LIN {X 0,Y 388.743,Z 625.918,A -85,B 0,C 180,E1 -11613.109,E2 -11613.109} C_VEL
LIN {X 0,Y 388.739,Z 624.507,A -85,B 0,C 180,E1 -11614.147,E2 -11614.147} C_VEL
LIN {X 0,Y 388.741,Z 621.416,A -85,B 0,C 180,E1 -11615.775,E2 -11615.775} C_VEL
LIN {X 0,Y 388.932,Z 617.582,A -85,B 0,C 180,E1 -11617.267,E2 -11617.267} C_VEL
LIN {X 0,Y 389.218,Z 612.461,A -85,B 0,C 180,E1 -11618.829,E2 -11618.829} C_VEL
LIN {X 0,Y 389.638,Z 606.07,A -85,B 0,C 180,E1 -11620.392,E2 -11620.392} C_VEL
LIN {X 0,Y 390.339,Z 598.224,A -85,B 0,C 180,E1 -11621.95,E2 -11621.95} C_VEL
LIN {X 0,Y 391.121,Z 588.53,A -85,B 0,C 180,E1 -11623.509,E2 -11623.509} C_VEL
LIN {X 0,Y 392.289,Z 577.655,A -85,B 0,C 180,E1 -11624.924,E2 -11624.924} C_VEL
LIN {X 0,Y 393.398,Z 566.699,A -85,B 0,C 180,E1 -11626.076,E2 -11626.076} C_VEL
LIN {X 0,Y 394.452,Z 554.774,A -85,B 0,C 180,E1 -11627.097,E2 -11627.097} C_VEL
LIN {X 0,Y 393.842,Z 541.578,A -85,B 0,C 180,E1 -11628.085,E2 -11628.085} C_VEL
LIN {X 0,Y 392.175,Z 529.359,A -85,B 0,C 180,E1 -11628.886,E2 -11628.886} C_VEL
LIN {X 0,Y 389.451,Z 517.138,A -85,B 0,C 180,E1 -11629.64,E2 -11629.64} C_VEL
LIN {X 0,Y 389.818,Z 510.265,A -85,B 0,C 180,E1 -11632.714,E2 -11632.714} C_VEL
LIN {X 0,Y 390.359,Z 503.675,A -85,B 0,C 180,E1 -11635.816,E2 -11635.816} C_VEL
LIN {X 0,Y 391.097,Z 496.234,A -85,B 0,C 180,E1 -11639.615,E2 -11639.615} C_VEL
LIN {X 0,Y 391.871,Z 491.031,A -85,B 0,C 180,E1 -11642.55,E2 -11642.55} C_VEL
LIN {X 0,Y 392.449,Z 487.212,A -85,B 0,C 180,E1 -11644.964,E2 -11644.964} C_VEL
LIN {X 0,Y 392.679,Z 485.233,A -85,B 0,C 180,E1 -11646.352,E2 -11646.352} C_VEL
LIN {X 0,Y 392.542,Z 482.258,A -85,B 0,C 180,E1 -11648.802,E2 -11648.802} C_VEL
LIN {X 0,Y 392.126,Z 479.631,A -85,B 0,C 180,E1 -11651.54,E2 -11651.54} C_VEL
LIN {X 0,Y 391.771,Z 477.585,A -85,B 0,C 180,E1 -11654.397,E2 -11654.397} C_VEL
LIN {X 0,Y 391.509,Z 476.207,A -85,B 0,C 180,E1 -11657.391,E2 -11657.391} C_VEL
LIN {X 0,Y 391.301,Z 475.518,A -85,B 0,C 180,E1 -11660.562,E2 -11660.562} C_VEL
LIN {X 0,Y 391.175,Z 475.523,A -85,B 0,C 180,E1 -11663.638,E2 -11663.638} C_VEL
LIN {X 0,Y 390.977,Z 475.957,A -85,B 0,C 180,E1 -11666.135,E2 -11666.135} C_VEL
LIN {X 0,Y 390.563,Z 477.165,A -85,B 0,C 180,E1 -11669.745,E2 -11669.745} C_VEL
LIN {X 0,Y 390.158,Z 478.822,A -85,B 0,C 180,E1 -11673.235,E2 -11673.235} C_VEL
LIN {X 0,Y 389.91,Z 480.896,A -85,B 0,C 180,E1 -11676.819,E2 -11676.819} C_VEL
LIN {X 0,Y 389.699,Z 483.382,A -85,B 0,C 180,E1 -11680.549,E2 -11680.549} C_VEL
LIN {X 0,Y 394.387,Z 496.846,A -85,B 0,C 180,E1 -11681.609,E2 -11681.609} C_VEL
LIN {X 0,Y 396.401,Z 504.348,A -85,B 0,C 180,E1 -11682.226,E2 -11682.226} C_VEL
LIN {X 0,Y 396.513,Z 507.54,A -85,B 0,C 180,E1 -11682.463,E2 -11682.463} C_VEL
LIN {X 0,Y 395.554,Z 519.166,A -85,B 0,C 180,E1 -11683.352,E2 -11683.352} C_VEL
LIN {X 0,Y 394.437,Z 530.942,A -85,B 0,C 180,E1 -11684.498,E2 -11684.498} C_VEL
LIN {X 0,Y 393.337,Z 541.589,A -85,B 0,C 180,E1 -11685.778,E2 -11685.778} C_VEL
LIN {X 0,Y 392.489,Z 548.688,A -85,B 0,C 180,E1 -11686.803,E2 -11686.803} C_VEL
LIN {X 0,Y 391.496,Z 557.528,A -85,B 0,C 180,E1 -11688.349,E2 -11688.349} C_VEL
LIN {X 0,Y 390.789,Z 564.646,A -85,B 0,C 180,E1 -11689.901,E2 -11689.901} C_VEL
LIN {X 0,Y 390.054,Z 571.233,A -85,B 0,C 180,E1 -11691.712,E2 -11691.712} C_VEL
LIN {X 0,Y 389.636,Z 575.213,A -85,B 0,C 180,E1 -11693.115,E2 -11693.115} C_VEL
LIN {X 0,Y 389.321,Z 578.854,A -85,B 0,C 180,E1 -11694.822,E2 -11694.822} C_VEL
LIN {X 0,Y 389.232,Z 580.45,A -85,B 0,C 180,E1 -11695.858,E2 -11695.858} C_VEL
LIN {X 0,Y 389.059,Z 581.651,A -85,B 0,C 180,E1 -11696.894,E2 -11696.894} C_VEL
LIN {X 0,Y 388.959,Z 582.45,A -85,B 0,C 180,E1 -11697.929,E2 -11697.929} C_VEL
LIN {X 0,Y 388.866,Z 582.808,A -85,B 0,C 180,E1 -11698.965,E2 -11698.965} C_VEL
LIN {X 0,Y 388.812,Z 582.757,A -85,B 0,C 180,E1 -11700,E2 -11700} C_VEL
LIN {X 0,Y 388.817,Z 582.311,A -85,B 0,C 180,E1 -11701.036,E2 -11701.036} C_VEL
LIN {X 0,Y 388.9,Z 581.459,A -85,B 0,C 180,E1 -11702.072,E2 -11702.072} C_VEL
LIN {X 0,Y 388.979,Z 580.155,A -85,B 0,C 180,E1 -11703.107,E2 -11703.107} C_VEL
LIN {X 0,Y 388.992,Z 577.422,A -85,B 0,C 180,E1 -11704.664,E2 -11704.664} C_VEL
LIN {X 0,Y 389.28,Z 572.842,A -85,B 0,C 180,E1 -11706.498,E2 -11706.498} C_VEL
LIN {X 0,Y 389.595,Z 566.823,A -85,B 0,C 180,E1 -11708.298,E2 -11708.298} C_VEL
LIN {X 0,Y 390.104,Z 560.131,A -85,B 0,C 180,E1 -11709.855,E2 -11709.855} C_VEL
LIN {X 0,Y 390.663,Z 551.845,A -85,B 0,C 180,E1 -11711.414,E2 -11711.414} C_VEL
LIN {X 0,Y 391.294,Z 543.426,A -85,B 0,C 180,E1 -11712.711,E2 -11712.711} C_VEL
LIN {X 0,Y 392.117,Z 533.146,A -85,B 0,C 180,E1 -11714.003,E2 -11714.003} C_VEL
LIN {X 0,Y 392.805,Z 521.468,A -85,B 0,C 180,E1 -11715.191,E2 -11715.191} C_VEL
LIN {X 0,Y 393.462,Z 510.623,A -85,B 0,C 180,E1 -11716.073,E2 -11716.073} C_VEL
LIN {X 0,Y 393.827,Z 501.011,A -85,B 0,C 180,E1 -11716.706,E2 -11716.706} C_VEL
LIN {X 0,Y 391.065,Z 488.304,A -85,B 0,C 180,E1 -11717.466,E2 -11717.466} C_VEL
LIN {X 0,Y 388.963,Z 478.596,A -85,B 0,C 180,E1 -11717.923,E2 -11717.923} C_VEL
LIN {X 0,Y 389.004,Z 475.238,A -85,B 0,C 180,E1 -11721.182,E2 -11721.182} C_VEL
LIN {X 0,Y 389.069,Z 471.846,A -85,B 0,C 180,E1 -11724.549,E2 -11724.549} C_VEL
LIN {X 0,Y 389.216,Z 468.447,A -85,B 0,C 180,E1 -11728.001,E2 -11728.001} C_VEL
LIN {X 0,Y 389.39,Z 467.987,A -85,B 0,C 180,E1 -11729.963,E2 -11729.963} C_VEL
LIN {X 0,Y 389.666,Z 467.948,A -85,B 0,C 180,E1 -11732.758,E2 -11732.758} C_VEL
LIN {X 0,Y 389.974,Z 467.908,A -85,B 0,C 180,E1 -11735.808,E2 -11735.808} C_VEL
LIN {X 0,Y 390.07,Z 467.894,A -85,B 0,C 180,E1 -11739.218,E2 -11739.218} C_VEL
LIN {X 0,Y 390.049,Z 467.9,A -85,B 0,C 180,E1 -11742.375,E2 -11742.375} C_VEL
LIN {X 0,Y 390.05,Z 467.897,A -85,B 0,C 180,E1 -11745.355,E2 -11745.355} C_VEL
LIN {X 0,Y 390.036,Z 467.902,A -85,B 0,C 180,E1 -11748.187,E2 -11748.187} C_VEL
LIN {X 0,Y 390.097,Z 467.891,A -85,B 0,C 180,E1 -11750.908,E2 -11750.908} C_VEL
LIN {X 0,Y 390.089,Z 467.892,A -85,B 0,C 180,E1 -11754.793,E2 -11754.793} C_VEL
LIN {X 0,Y 390.036,Z 467.902,A -85,B 0,C 180,E1 -11757.875,E2 -11757.875} C_VEL
LIN {X 0,Y 390.063,Z 467.896,A -85,B 0,C 180,E1 -11760.891,E2 -11760.891} C_VEL
LIN {X 0,Y 390.124,Z 467.893,A -85,B 0,C 180,E1 -11764.257,E2 -11764.257} C_VEL
LIN {X 0,Y 390.045,Z 467.9,A -85,B 0,C 180,E1 -11767.766,E2 -11767.766} C_VEL
LIN {X 0,Y 390.11,Z 467.89,A -85,B 0,C 180,E1 -11771.078,E2 -11771.078} C_VEL
LIN {X 0,Y 390.144,Z 467.889,A -85,B 0,C 180,E1 -11774.323,E2 -11774.323} C_VEL
LIN {X 0,Y 390.176,Z 467.882,A -85,B 0,C 180,E1 -11777.517,E2 -11777.517} C_VEL
LIN {X 0,Y 390.32,Z 467.866,A -85,B 0,C 180,E1 -11781.718,E2 -11781.718} C_VEL
LIN {X 0,Y 390.335,Z 467.865,A -85,B 0,C 180,E1 -11783.798,E2 -11783.798} C_VEL
LIN {X 0,Y 390.423,Z 467.853,A -85,B 0,C 180,E1 -11787.937,E2 -11787.937} C_VEL
LIN {X 0,Y 390.554,Z 467.838,A -85,B 0,C 180,E1 -11790,E2 -11790} C_VEL
LIN {X 0,Y 390.315,Z 467.863,A -85,B 0,C 180,E1 -11793.097,E2 -11793.097} C_VEL
LIN {X 0,Y 390.304,Z 467.868,A -85,B 0,C 180,E1 -11796.202,E2 -11796.202} C_VEL
LIN {X 0,Y 390.198,Z 467.88,A -85,B 0,C 180,E1 -11799.329,E2 -11799.329} C_VEL
LIN {X 0,Y 390.176,Z 467.882,A -85,B 0,C 180,E1 -11802.483,E2 -11802.483} C_VEL
LIN {X 0,Y 390.145,Z 467.888,A -85,B 0,C 180,E1 -11805.677,E2 -11805.677} C_VEL
LIN {X 0,Y 390.111,Z 467.89,A -85,B 0,C 180,E1 -11808.922,E2 -11808.922} C_VEL
LIN {X 0,Y 390.041,Z 467.9,A -85,B 0,C 180,E1 -11812.32,E2 -11812.32} C_VEL
LIN {X 0,Y 390.123,Z 467.891,A -85,B 0,C 180,E1 -11815.743,E2 -11815.743} C_VEL
LIN {X 0,Y 390.115,Z 467.887,A -85,B 0,C 180,E1 -11816.807,E2 -11816.807} C_VEL
LIN {X 0,Y 389.411,Z 467.98,A -85,B 0,C 180,E1 -11817.668,E2 -11817.668} C_VEL
LIN {X 0,Y 386.517,Z 468.337,A -85,B 0,C 180,E1 -11819.069,E2 -11819.069} C_VEL
LIN {X 0,Y 384.091,Z 468.642,A -85,B 0,C 180,E1 -11820.2,E2 -11820.2} C_VEL
LIN {X 0,Y 383.057,Z 468.768,A -85,B 0,C 180,E1 -11821.076,E2 -11821.076} C_VEL
LIN {X 0,Y 382.977,Z 468.777,A -85,B 0,C 180,E1 -11821.372,E2 -11821.372} C_VEL
LIN {X 0,Y 383.023,Z 468.772,A -85,B 0,C 180,E1 -11824.668,E2 -11824.668} C_VEL
LIN {X 0,Y 383.006,Z 468.778,A -85,B 0,C 180,E1 -11827.904,E2 -11827.904} C_VEL
LIN {X 0,Y 382.989,Z 468.778,A -85,B 0,C 180,E1 -11831.347,E2 -11831.347} C_VEL
LIN {X 0,Y 383.001,Z 468.777,A -85,B 0,C 180,E1 -11834.303,E2 -11834.303} C_VEL
LIN {X 0,Y 383.014,Z 468.775,A -85,B 0,C 180,E1 -11837.24,E2 -11837.24} C_VEL
LIN {X 0,Y 383.018,Z 468.772,A -85,B 0,C 180,E1 -11840.413,E2 -11840.413} C_VEL
LIN {X 0,Y 382.973,Z 468.78,A -85,B 0,C 180,E1 -11844.038,E2 -11844.038} C_VEL
LIN {X 0,Y 382.774,Z 468.804,A -85,B 0,C 180,E1 -11846.576,E2 -11846.576} C_VEL
LIN {X 0,Y 382.417,Z 468.852,A -85,B 0,C 180,E1 -11849.742,E2 -11849.742} C_VEL
LIN {X 0,Y 382.061,Z 468.898,A -85,B 0,C 180,E1 -11852.621,E2 -11852.621} C_VEL
LIN {X 0,Y 381.965,Z 469.45,A -85,B 0,C 180,E1 -11853.794,E2 -11853.794} C_VEL
LIN {X 0,Y 381.906,Z 473.282,A -85,B 0,C 180,E1 -11857.266,E2 -11857.266} C_VEL
LIN {X 0,Y 381.87,Z 477.054,A -85,B 0,C 180,E1 -11860.653,E2 -11860.653} C_VEL
LIN {X 0,Y 381.871,Z 478.605,A -85,B 0,C 180,E1 -11861.963,E2 -11861.963} C_VEL
LIN {X 0,Y 384.636,Z 491.634,A -85,B 0,C 180,E1 -11862.594,E2 -11862.594} C_VEL
LIN {X 0,Y 386.939,Z 502.891,A -85,B 0,C 180,E1 -11863.309,E2 -11863.309} C_VEL
LIN {X 0,Y 386.237,Z 514.849,A -85,B 0,C 180,E1 -11864.16,E2 -11864.16} C_VEL
LIN {X 0,Y 385.572,Z 526.535,A -85,B 0,C 180,E1 -11865.215,E2 -11865.215} C_VEL
LIN {X 0,Y 384.771,Z 537.046,A -85,B 0,C 180,E1 -11866.398,E2 -11866.398} C_VEL
LIN {X 0,Y 383.944,Z 547.495,A -85,B 0,C 180,E1 -11867.848,E2 -11867.848} C_VEL
LIN {X 0,Y 383.25,Z 556.654,A -85,B 0,C 180,E1 -11869.433,E2 -11869.433} C_VEL
LIN {X 0,Y 382.693,Z 564.046,A -85,B 0,C 180,E1 -11871.019,E2 -11871.019} C_VEL
LIN {X 0,Y 382.348,Z 570,A -85,B 0,C 180,E1 -11872.607,E2 -11872.607} C_VEL
LIN {X 0,Y 382.089,Z 574.685,A -85,B 0,C 180,E1 -11874.193,E2 -11874.193} C_VEL
LIN {X 0,Y 381.872,Z 578.249,A -85,B 0,C 180,E1 -11875.778,E2 -11875.778} C_VEL
LIN {X 0,Y 381.88,Z 580.026,A -85,B 0,C 180,E1 -11876.835,E2 -11876.835} C_VEL
LIN {X 0,Y 381.827,Z 581.4,A -85,B 0,C 180,E1 -11877.89,E2 -11877.89} C_VEL
LIN {X 0,Y 381.737,Z 582.371,A -85,B 0,C 180,E1 -11878.945,E2 -11878.945} C_VEL
LIN {X 0,Y 381.727,Z 582.881,A -85,B 0,C 180,E1 -11880,E2 -11880} C_VEL
LIN {X 0,Y 381.771,Z 582.992,A -85,B 0,C 180,E1 -11881.055,E2 -11881.055} C_VEL
LIN {X 0,Y 381.875,Z 582.707,A -85,B 0,C 180,E1 -11882.109,E2 -11882.109} C_VEL
LIN {X 0,Y 382.006,Z 581.987,A -85,B 0,C 180,E1 -11883.164,E2 -11883.164} C_VEL
LIN {X 0,Y 382.177,Z 580.837,A -85,B 0,C 180,E1 -11884.218,E2 -11884.218} C_VEL
LIN {X 0,Y 382.189,Z 579.305,A -85,B 0,C 180,E1 -11885.275,E2 -11885.275} C_VEL
LIN {X 0,Y 382.572,Z 576.053,A -85,B 0,C 180,E1 -11886.903,E2 -11886.903} C_VEL
LIN {X 0,Y 382.999,Z 571.944,A -85,B 0,C 180,E1 -11888.441,E2 -11888.441} C_VEL
LIN {X 0,Y 383.807,Z 565.49,A -85,B 0,C 180,E1 -11890.284,E2 -11890.284} C_VEL
LIN {X 0,Y 384.51,Z 558.499,A -85,B 0,C 180,E1 -11891.866,E2 -11891.866} C_VEL
LIN {X 0,Y 385.567,Z 549.85,A -85,B 0,C 180,E1 -11893.438,E2 -11893.438} C_VEL
LIN {X 0,Y 386.583,Z 541.045,A -85,B 0,C 180,E1 -11894.745,E2 -11894.745} C_VEL
LIN {X 0,Y 387.837,Z 530.124,A -85,B 0,C 180,E1 -11896.065,E2 -11896.065} C_VEL
LIN {X 0,Y 389.023,Z 518.194,A -85,B 0,C 180,E1 -11897.207,E2 -11897.207} C_VEL
LIN {X 0,Y 389.929,Z 506.361,A -85,B 0,C 180,E1 -11898.116,E2 -11898.116} C_VEL
LIN {X 0,Y 387.401,Z 496.099,A -85,B 0,C 180,E1 -11898.999,E2 -11898.999} C_VEL
LIN {X 0,Y 383.296,Z 484.971,A -85,B 0,C 180,E1 -11899.92,E2 -11899.92} C_VEL
LIN {X 0,Y 382.567,Z 482.635,A -85,B 0,C 180,E1 -11900.107,E2 -11900.107} C_VEL
LIN {X 0,Y 382.645,Z 478.78,A -85,B 0,C 180,E1 -11903.833,E2 -11903.833} C_VEL
LIN {X 0,Y 382.729,Z 476.402,A -85,B 0,C 180,E1 -11906.149,E2 -11906.149} C_VEL
LIN {X 0,Y 382.822,Z 472.719,A -85,B 0,C 180,E1 -11909.714,E2 -11909.714} C_VEL
LIN {X 0,Y 382.879,Z 470.008,A -85,B 0,C 180,E1 -11912.396,E2 -11912.396} C_VEL
LIN {X 0,Y 382.808,Z 469.012,A -85,B 0,C 180,E1 -11913.42,E2 -11913.42} C_VEL
LIN {X 0,Y 382.987,Z 468.78,A -85,B 0,C 180,E1 -11916.155,E2 -11916.155} C_VEL
LIN {X 0,Y 383.017,Z 468.778,A -85,B 0,C 180,E1 -11919.587,E2 -11919.587} C_VEL
LIN {X 0,Y 383.006,Z 468.777,A -85,B 0,C 180,E1 -11922.778,E2 -11922.778} C_VEL
LIN {X 0,Y 383.057,Z 468.821,A -85,B 0,C 180,E1 -11926.355,E2 -11926.355} C_VEL
LIN {X 0,Y 384.052,Z 474.383,A -85,B 0,C 180,E1 -11929.486,E2 -11929.486} C_VEL
LIN {X 0,Y 385.125,Z 480.888,A -85,B 0,C 180,E1 -11932.972,E2 -11932.972} C_VEL
LIN {X 0,Y 385.096,Z 485.339,A -85,B 0,C 180,E1 -11935.21,E2 -11935.21} C_VEL
LIN {X 0,Y 384.35,Z 492.339,A -85,B 0,C 180,E1 -11938.591,E2 -11938.591} C_VEL
LIN {X 0,Y 383.676,Z 499.918,A -85,B 0,C 180,E1 -11942.154,E2 -11942.154} C_VEL
LIN {X 0,Y 383.037,Z 507.462,A -85,B 0,C 180,E1 -11945.617,E2 -11945.617} C_VEL
LIN {X 0,Y 382.543,Z 514.974,A -85,B 0,C 180,E1 -11949.007,E2 -11949.007} C_VEL
LIN {X 0,Y 382.39,Z 517.633,A -85,B 0,C 180,E1 -11950.192,E2 -11950.192} C_VEL
LIN {X 0,Y 385.614,Z 533.963,A -85,B 0,C 180,E1 -11951.245,E2 -11951.245} C_VEL
LIN {X 0,Y 386.776,Z 546.578,A -85,B 0,C 180,E1 -11952.144,E2 -11952.144} C_VEL
LIN {X 0,Y 387.184,Z 556.631,A -85,B 0,C 180,E1 -11952.981,E2 -11952.981} C_VEL
LIN {X 0,Y 386.052,Z 567.959,A -85,B 0,C 180,E1 -11954.017,E2 -11954.017} C_VEL
LIN {X 0,Y 384.872,Z 579.687,A -85,B 0,C 180,E1 -11955.356,E2 -11955.356} C_VEL
LIN {X 0,Y 383.891,Z 589.69,A -85,B 0,C 180,E1 -11956.771,E2 -11956.771} C_VEL
LIN {X 0,Y 383.004,Z 598.767,A -85,B 0,C 180,E1 -11958.355,E2 -11958.355} C_VEL
LIN {X 0,Y 382.388,Z 606.219,A -85,B 0,C 180,E1 -11959.944,E2 -11959.944} C_VEL
LIN {X 0,Y 382.02,Z 612.209,A -85,B 0,C 180,E1 -11961.537,E2 -11961.537} C_VEL
LIN {X 0,Y 381.745,Z 618.814,A -85,B 0,C 180,E1 -11963.801,E2 -11963.801} C_VEL
LIN {X 0,Y 381.747,Z 622.148,A -85,B 0,C 180,E1 -11965.248,E2 -11965.248} C_VEL
LIN {X 0,Y 381.688,Z 624.791,A -85,B 0,C 180,E1 -11966.833,E2 -11966.833} C_VEL
LIN {X 0,Y 381.779,Z 626.012,A -85,B 0,C 180,E1 -11967.89,E2 -11967.89} C_VEL
LIN {X 0,Y 381.739,Z 626.785,A -85,B 0,C 180,E1 -11968.945,E2 -11968.945} C_VEL
LIN {X 0,Y 381.736,Z 627.103,A -85,B 0,C 180,E1 -11970,E2 -11970} C_VEL
LIN {X 0,Y 381.731,Z 627.012,A -85,B 0,C 180,E1 -11971.055,E2 -11971.055} C_VEL
LIN {X 0,Y 381.756,Z 626.514,A -85,B 0,C 180,E1 -11972.11,E2 -11972.11} C_VEL
LIN {X 0,Y 381.646,Z 625.564,A -85,B 0,C 180,E1 -11973.167,E2 -11973.167} C_VEL
LIN {X 0,Y 381.662,Z 624.175,A -85,B 0,C 180,E1 -11974.224,E2 -11974.224} C_VEL
LIN {X 0,Y 381.693,Z 620.602,A -85,B 0,C 180,E1 -11976.127,E2 -11976.127} C_VEL
LIN {X 0,Y 381.937,Z 615.822,A -85,B 0,C 180,E1 -11977.933,E2 -11977.933} C_VEL
LIN {X 0,Y 382.36,Z 609.307,A -85,B 0,C 180,E1 -11979.789,E2 -11979.789} C_VEL
LIN {X 0,Y 382.939,Z 602.299,A -85,B 0,C 180,E1 -11981.379,E2 -11981.379} C_VEL
LIN {X 0,Y 383.775,Z 593.737,A -85,B 0,C 180,E1 -11982.964,E2 -11982.964} C_VEL
LIN {X 0,Y 384.666,Z 584.669,A -85,B 0,C 180,E1 -11984.336,E2 -11984.336} C_VEL
LIN {X 0,Y 385.946,Z 573.519,A -85,B 0,C 180,E1 -11985.716,E2 -11985.716} C_VEL
LIN {X 0,Y 387.25,Z 561.84,A -85,B 0,C 180,E1 -11986.881,E2 -11986.881} C_VEL
LIN {X 0,Y 387.697,Z 554.173,A -85,B 0,C 180,E1 -11987.54,E2 -11987.54} C_VEL
LIN {X 0,Y 387.066,Z 540.9,A -85,B 0,C 180,E1 -11988.569,E2 -11988.569} C_VEL
LIN {X 0,Y 385.33,Z 529.072,A -85,B 0,C 180,E1 -11989.391,E2 -11989.391} C_VEL
LIN {X 0,Y 382.474,Z 516.569,A -85,B 0,C 180,E1 -11990.191,E2 -11990.191} C_VEL
LIN {X 0,Y 382.931,Z 508.781,A -85,B 0,C 180,E1 -11993.814,E2 -11993.814} C_VEL
LIN {X 0,Y 383.556,Z 501.826,A -85,B 0,C 180,E1 -11997.264,E2 -11997.264} C_VEL
LIN {X 0,Y 384.247,Z 496.405,A -85,B 0,C 180,E1 -12000.178,E2 -12000.178} C_VEL
LIN {X 0,Y 385.024,Z 491.301,A -85,B 0,C 180,E1 -12003.203,E2 -12003.203} C_VEL
LIN {X 0,Y 385.577,Z 487.602,A -85,B 0,C 180,E1 -12005.681,E2 -12005.681} C_VEL
LIN {X 0,Y 385.743,Z 485.902,A -85,B 0,C 180,E1 -12006.959,E2 -12006.959} C_VEL
LIN {X 0,Y 385.677,Z 484.182,A -85,B 0,C 180,E1 -12008.412,E2 -12008.412} C_VEL
LIN {X 0,Y 385.195,Z 481.144,A -85,B 0,C 180,E1 -12011.578,E2 -12011.578} C_VEL
LIN {X 0,Y 384.824,Z 479.04,A -85,B 0,C 180,E1 -12014.581,E2 -12014.581} C_VEL
LIN {X 0,Y 384.587,Z 477.73,A -85,B 0,C 180,E1 -12017.457,E2 -12017.457} C_VEL
LIN {X 0,Y 384.373,Z 477.075,A -85,B 0,C 180,E1 -12020.212,E2 -12020.212} C_VEL
LIN {X 0,Y 384.25,Z 476.956,A -85,B 0,C 180,E1 -12023.588,E2 -12023.588} C_VEL
LIN {X 0,Y 383.928,Z 477.492,A -85,B 0,C 180,E1 -12026.69,E2 -12026.69} C_VEL
LIN {X 0,Y 383.631,Z 478.356,A -85,B 0,C 180,E1 -12029.432,E2 -12029.432} C_VEL
LIN {X 0,Y 383.22,Z 479.79,A -85,B 0,C 180,E1 -12032.711,E2 -12032.711} C_VEL
LIN {X 0,Y 382.928,Z 481.668,A -85,B 0,C 180,E1 -12036.186,E2 -12036.186} C_VEL
LIN {X 0,Y 382.708,Z 484.076,A -85,B 0,C 180,E1 -12039.983,E2 -12039.983} C_VEL
LIN {X 0,Y 383.889,Z 487.251,A -85,B 0,C 180,E1 -12040.241,E2 -12040.241} C_VEL
LIN {X 0,Y 387.823,Z 498.174,A -85,B 0,C 180,E1 -12041.168,E2 -12041.168} C_VEL
LIN {X 0,Y 390.025,Z 506.66,A -85,B 0,C 180,E1 -12041.923,E2 -12041.923} C_VEL
LIN {X 0,Y 389.07,Z 519.608,A -85,B 0,C 180,E1 -12042.931,E2 -12042.931} C_VEL
LIN {X 0,Y 387.943,Z 530.793,A -85,B 0,C 180,E1 -12044.029,E2 -12044.029} C_VEL
LIN {X 0,Y 386.756,Z 541.014,A -85,B 0,C 180,E1 -12045.262,E2 -12045.262} C_VEL
LIN {X 0,Y 385.675,Z 549.862,A -85,B 0,C 180,E1 -12046.565,E2 -12046.565} C_VEL
LIN {X 0,Y 384.632,Z 558.519,A -85,B 0,C 180,E1 -12048.138,E2 -12048.138} C_VEL
LIN {X 0,Y 383.858,Z 565.557,A -85,B 0,C 180,E1 -12049.717,E2 -12049.717} C_VEL
LIN {X 0,Y 383.313,Z 570.338,A -85,B 0,C 180,E1 -12051.034,E2 -12051.034} C_VEL
LIN {X 0,Y 382.729,Z 574.975,A -85,B 0,C 180,E1 -12052.615,E2 -12052.615} C_VEL
LIN {X 0,Y 382.377,Z 577.475,A -85,B 0,C 180,E1 -12053.669,E2 -12053.669} C_VEL
LIN {X 0,Y 382.265,Z 579.466,A -85,B 0,C 180,E1 -12054.726,E2 -12054.726} C_VEL
LIN {X 0,Y 382.191,Z 581.026,A -85,B 0,C 180,E1 -12055.782,E2 -12055.782} C_VEL
LIN {X 0,Y 382.007,Z 582.197,A -85,B 0,C 180,E1 -12056.836,E2 -12056.836} C_VEL
LIN {X 0,Y 381.892,Z 582.954,A -85,B 0,C 180,E1 -12057.891,E2 -12057.891} C_VEL
LIN {X 0,Y 381.793,Z 583.266,A -85,B 0,C 180,E1 -12058.945,E2 -12058.945} C_VEL
LIN {X 0,Y 381.738,Z 583.18,A -85,B 0,C 180,E1 -12060,E2 -12060} C_VEL
LIN {X 0,Y 381.747,Z 582.697,A -85,B 0,C 180,E1 -12061.055,E2 -12061.055} C_VEL
LIN {X 0,Y 381.836,Z 581.785,A -85,B 0,C 180,E1 -12062.11,E2 -12062.11} C_VEL
LIN {X 0,Y 381.885,Z 580.439,A -85,B 0,C 180,E1 -12063.165,E2 -12063.165} C_VEL
LIN {X 0,Y 381.927,Z 577.632,A -85,B 0,C 180,E1 -12064.75,E2 -12064.75} C_VEL
LIN {X 0,Y 382.171,Z 573.779,A -85,B 0,C 180,E1 -12066.335,E2 -12066.335} C_VEL
LIN {X 0,Y 382.43,Z 568.78,A -85,B 0,C 180,E1 -12067.923,E2 -12067.923} C_VEL
LIN {X 0,Y 382.896,Z 562.497,A -85,B 0,C 180,E1 -12069.509,E2 -12069.509} C_VEL
LIN {X 0,Y 383.463,Z 554.714,A -85,B 0,C 180,E1 -12071.096,E2 -12071.096} C_VEL
LIN {X 0,Y 384.187,Z 544.983,A -85,B 0,C 180,E1 -12072.681,E2 -12072.681} C_VEL
LIN {X 0,Y 385.01,Z 535.04,A -85,B 0,C 180,E1 -12073.997,E2 -12073.997} C_VEL
LIN {X 0,Y 385.659,Z 524.731,A -85,B 0,C 180,E1 -12075.109,E2 -12075.109} C_VEL
LIN {X 0,Y 386.4,Z 513.282,A -85,B 0,C 180,E1 -12076.104,E2 -12076.104} C_VEL
LIN {X 0,Y 386.954,Z 502.925,A -85,B 0,C 180,E1 -12076.826,E2 -12076.826} C_VEL
LIN {X 0,Y 384.666,Z 491.668,A -85,B 0,C 180,E1 -12077.543,E2 -12077.543} C_VEL
LIN {X 0,Y 381.902,Z 478.925,A -85,B 0,C 180,E1 -12078.194,E2 -12078.194} C_VEL
LIN {X 0,Y 381.947,Z 475.455,A -85,B 0,C 180,E1 -12081.593,E2 -12081.593} C_VEL
LIN {X 0,Y 382.041,Z 472.023,A -85,B 0,C 180,E1 -12085.031,E2 -12085.031} C_VEL
LIN {X 0,Y 382.176,Z 469.103,A -85,B 0,C 180,E1 -12088.03,E2 -12088.03} C_VEL
LIN {X 0,Y 382.44,Z 468.848,A -85,B 0,C 180,E1 -12090.968,E2 -12090.968} C_VEL
LIN {X 0,Y 382.812,Z 468.801,A -85,B 0,C 180,E1 -12094.69,E2 -12094.69} C_VEL
LIN {X 0,Y 382.982,Z 468.777,A -85,B 0,C 180,E1 -12097.271,E2 -12097.271} C_VEL
LIN {X 0,Y 383.011,Z 468.776,A -85,B 0,C 180,E1 -12099.959,E2 -12099.959} C_VEL
LIN {X 0,Y 383.009,Z 468.775,A -85,B 0,C 180,E1 -12102.779,E2 -12102.779} C_VEL
LIN {X 0,Y 383.002,Z 468.777,A -85,B 0,C 180,E1 -12105.79,E2 -12105.79} C_VEL
LIN {X 0,Y 382.993,Z 468.777,A -85,B 0,C 180,E1 -12108.796,E2 -12108.796} C_VEL
LIN {X 0,Y 383.006,Z 468.778,A -85,B 0,C 180,E1 -12112.096,E2 -12112.096} C_VEL
LIN {X 0,Y 383.022,Z 468.772,A -85,B 0,C 180,E1 -12115.332,E2 -12115.332} C_VEL
LIN {X 0,Y 382.987,Z 468.777,A -85,B 0,C 180,E1 -12119.082,E2 -12119.082} C_VEL
LIN {X 0,Y 383.061,Z 468.769,A -85,B 0,C 180,E1 -12122.698,E2 -12122.698} C_VEL
LIN {X 0,Y 383.038,Z 468.775,A -85,B 0,C 180,E1 -12126.193,E2 -12126.193} C_VEL
LIN {X 0,Y 383.06,Z 468.769,A -85,B 0,C 180,E1 -12129.599,E2 -12129.599} C_VEL
LIN {X 0,Y 383.11,Z 468.762,A -85,B 0,C 180,E1 -12132.931,E2 -12132.931} C_VEL
LIN {X 0,Y 383.13,Z 468.761,A -85,B 0,C 180,E1 -12136.464,E2 -12136.464} C_VEL
LIN {X 0,Y 383.156,Z 468.757,A -85,B 0,C 180,E1 -12140.498,E2 -12140.498} C_VEL
LIN {X 0,Y 383.279,Z 468.742,A -85,B 0,C 180,E1 -12142.625,E2 -12142.625} C_VEL
LIN {X 0,Y 383.204,Z 468.75,A -85,B 0,C 180,E1 -12144.739,E2 -12144.739} C_VEL
LIN {X 0,Y 383.391,Z 468.729,A -85,B 0,C 180,E1 -12147.899,E2 -12147.899} C_VEL
LIN {X 0,Y 383.523,Z 468.714,A -85,B 0,C 180,E1 -12150,E2 -12150} C_VEL
LIN {X 0,Y 383.251,Z 468.743,A -85,B 0,C 180,E1 -12153.154,E2 -12153.154} C_VEL
LIN {X 0,Y 383.261,Z 468.746,A -85,B 0,C 180,E1 -12156.317,E2 -12156.317} C_VEL
LIN {X 0,Y 383.148,Z 468.759,A -85,B 0,C 180,E1 -12159.502,E2 -12159.502} C_VEL
LIN {X 0,Y 383.141,Z 468.757,A -85,B 0,C 180,E1 -12162.716,E2 -12162.716} C_VEL
LIN {X 0,Y 383.086,Z 468.768,A -85,B 0,C 180,E1 -12165.973,E2 -12165.973} C_VEL
LIN {X 0,Y 383.066,Z 468.768,A -85,B 0,C 180,E1 -12169.284,E2 -12169.284} C_VEL
LIN {X 0,Y 383,Z 468.775,A -85,B 0,C 180,E1 -12172.665,E2 -12172.665} C_VEL
LIN {X 0,Y 383.084,Z 468.767,A -85,B 0,C 180,E1 -12176.123,E2 -12176.123} C_VEL
LIN {X 0,Y 382.997,Z 468.78,A -85,B 0,C 180,E1 -12179.7,E2 -12179.7} C_VEL
LIN {X 0,Y 382.977,Z 468.777,A -85,B 0,C 180,E1 -12181.372,E2 -12181.372} C_VEL
LIN {X 0,Y 382.317,Z 468.863,A -85,B 0,C 180,E1 -12182.251,E2 -12182.251} C_VEL
LIN {X 0,Y 379.464,Z 469.219,A -85,B 0,C 180,E1 -12183.679,E2 -12183.679} C_VEL
LIN {X 0,Y 377.052,Z 469.517,A -85,B 0,C 180,E1 -12184.833,E2 -12184.833} C_VEL
LIN {X 0,Y 376.027,Z 469.647,A -85,B 0,C 180,E1 -12185.726,E2 -12185.726} C_VEL
LIN {X 0,Y 375.95,Z 469.652,A -85,B 0,C 180,E1 -12186.029,E2 -12186.029} C_VEL
LIN {X 0,Y 375.968,Z 469.653,A -85,B 0,C 180,E1 -12189.462,E2 -12189.462} C_VEL
LIN {X 0,Y 375.938,Z 469.656,A -85,B 0,C 180,E1 -12193.189,E2 -12193.189} C_VEL
LIN {X 0,Y 375.938,Z 469.655,A -85,B 0,C 180,E1 -12196.81,E2 -12196.81} C_VEL
LIN {X 0,Y 375.966,Z 469.65,A -85,B 0,C 180,E1 -12200.537,E2 -12200.537} C_VEL
LIN {X 0,Y 375.94,Z 469.658,A -85,B 0,C 180,E1 -12203.501,E2 -12203.501} C_VEL
LIN {X 0,Y 375.787,Z 469.678,A -85,B 0,C 180,E1 -12205.87,E2 -12205.87} C_VEL
LIN {X 0,Y 375.528,Z 469.707,A -85,B 0,C 180,E1 -12208.397,E2 -12208.397} C_VEL
LIN {X 0,Y 375.101,Z 469.765,A -85,B 0,C 180,E1 -12212.069,E2 -12212.069} C_VEL
LIN {X 0,Y 374.938,Z 469.786,A -85,B 0,C 180,E1 -12213.264,E2 -12213.264} C_VEL
LIN {X 0,Y 374.823,Z 472.103,A -85,B 0,C 180,E1 -12215.637,E2 -12215.637} C_VEL
LIN {X 0,Y 374.804,Z 475.958,A -85,B 0,C 180,E1 -12219.128,E2 -12219.128} C_VEL
LIN {X 0,Y 374.824,Z 478.829,A -85,B 0,C 180,E1 -12221.712,E2 -12221.712} C_VEL
LIN {X 0,Y 377.568,Z 492.039,A -85,B 0,C 180,E1 -12222.373,E2 -12222.373} C_VEL
LIN {X 0,Y 379.943,Z 503.687,A -85,B 0,C 180,E1 -12223.131,E2 -12223.131} C_VEL
LIN {X 0,Y 379.171,Z 517.15,A -85,B 0,C 180,E1 -12224.134,E2 -12224.134} C_VEL
LIN {X 0,Y 378.498,Z 528.383,A -85,B 0,C 180,E1 -12225.208,E2 -12225.208} C_VEL
LIN {X 0,Y 377.573,Z 539.66,A -85,B 0,C 180,E1 -12226.545,E2 -12226.545} C_VEL
LIN {X 0,Y 376.845,Z 548.86,A -85,B 0,C 180,E1 -12227.889,E2 -12227.889} C_VEL
LIN {X 0,Y 376.152,Z 557.83,A -85,B 0,C 180,E1 -12229.504,E2 -12229.504} C_VEL
LIN {X 0,Y 375.581,Z 565.104,A -85,B 0,C 180,E1 -12231.119,E2 -12231.119} C_VEL
LIN {X 0,Y 375.294,Z 570.025,A -85,B 0,C 180,E1 -12232.467,E2 -12232.467} C_VEL
LIN {X 0,Y 375.026,Z 574.812,A -85,B 0,C 180,E1 -12234.084,E2 -12234.084} C_VEL
LIN {X 0,Y 374.797,Z 578.464,A -85,B 0,C 180,E1 -12235.698,E2 -12235.698} C_VEL
LIN {X 0,Y 374.786,Z 580.296,A -85,B 0,C 180,E1 -12236.775,E2 -12236.775} C_VEL
LIN {X 0,Y 374.764,Z 581.707,A -85,B 0,C 180,E1 -12237.85,E2 -12237.85} C_VEL
LIN {X 0,Y 374.67,Z 582.722,A -85,B 0,C 180,E1 -12238.925,E2 -12238.925} C_VEL
LIN {X 0,Y 374.656,Z 583.289,A -85,B 0,C 180,E1 -12240,E2 -12240} C_VEL
LIN {X 0,Y 374.702,Z 583.434,A -85,B 0,C 180,E1 -12241.074,E2 -12241.074} C_VEL
LIN {X 0,Y 374.812,Z 583.184,A -85,B 0,C 180,E1 -12242.149,E2 -12242.149} C_VEL
LIN {X 0,Y 374.956,Z 582.531,A -85,B 0,C 180,E1 -12243.223,E2 -12243.223} C_VEL
LIN {X 0,Y 375.132,Z 581.426,A -85,B 0,C 180,E1 -12244.297,E2 -12244.297} C_VEL
LIN {X 0,Y 375.141,Z 579.939,A -85,B 0,C 180,E1 -12245.375,E2 -12245.375} C_VEL
LIN {X 0,Y 375.541,Z 576.905,A -85,B 0,C 180,E1 -12246.964,E2 -12246.964} C_VEL
LIN {X 0,Y 376.025,Z 572.715,A -85,B 0,C 180,E1 -12248.599,E2 -12248.599} C_VEL
LIN {X 0,Y 376.881,Z 566.382,A -85,B 0,C 180,E1 -12250.475,E2 -12250.475} C_VEL
LIN {X 0,Y 377.834,Z 558.276,A -85,B 0,C 180,E1 -12252.351,E2 -12252.351} C_VEL
LIN {X 0,Y 378.771,Z 551.093,A -85,B 0,C 180,E1 -12253.684,E2 -12253.684} C_VEL
LIN {X 0,Y 379.849,Z 542.434,A -85,B 0,C 180,E1 -12255.012,E2 -12255.012} C_VEL
LIN {X 0,Y 381.224,Z 531.178,A -85,B 0,C 180,E1 -12256.416,E2 -12256.416} C_VEL
LIN {X 0,Y 382.461,Z 520.253,A -85,B 0,C 180,E1 -12257.512,E2 -12257.512} C_VEL
LIN {X 0,Y 383.466,Z 508.047,A -85,B 0,C 180,E1 -12258.503,E2 -12258.503} C_VEL
LIN {X 0,Y 380.746,Z 497.261,A -85,B 0,C 180,E1 -12259.482,E2 -12259.482} C_VEL
LIN {X 0,Y 376.705,Z 486.367,A -85,B 0,C 180,E1 -12260.46,E2 -12260.46} C_VEL
LIN {X 0,Y 375.567,Z 483.229,A -85,B 0,C 180,E1 -12260.739,E2 -12260.739} C_VEL
LIN {X 0,Y 375.681,Z 479.628,A -85,B 0,C 180,E1 -12264.303,E2 -12264.303} C_VEL
LIN {X 0,Y 375.752,Z 477.238,A -85,B 0,C 180,E1 -12266.672,E2 -12266.672} C_VEL
LIN {X 0,Y 375.934,Z 473.608,A -85,B 0,C 180,E1 -12270.315,E2 -12270.315} C_VEL
LIN {X 0,Y 375.936,Z 471.217,A -85,B 0,C 180,E1 -12272.83,E2 -12272.83} C_VEL
LIN {X 0,Y 375.842,Z 469.67,A -85,B 0,C 180,E1 -12274.636,E2 -12274.636} C_VEL
LIN {X 0,Y 375.937,Z 469.658,A -85,B 0,C 180,E1 -12276.743,E2 -12276.743} C_VEL
LIN {X 0,Y 375.991,Z 469.651,A -85,B 0,C 180,E1 -12279.971,E2 -12279.971} C_VEL
LIN {X 0,Y 375.933,Z 469.659,A -85,B 0,C 180,E1 -12283.765,E2 -12283.765} C_VEL
LIN {X 0,Y 376.01,Z 469.765,A -85,B 0,C 180,E1 -12286.153,E2 -12286.153} C_VEL
LIN {X 0,Y 377.157,Z 476.17,A -85,B 0,C 180,E1 -12289.818,E2 -12289.818} C_VEL
LIN {X 0,Y 378.122,Z 482.121,A -85,B 0,C 180,E1 -12293.056,E2 -12293.056} C_VEL
LIN {X 0,Y 378.09,Z 485.664,A -85,B 0,C 180,E1 -12294.873,E2 -12294.873} C_VEL
LIN {X 0,Y 377.415,Z 491.873,A -85,B 0,C 180,E1 -12297.946,E2 -12297.946} C_VEL
LIN {X 0,Y 376.763,Z 498.716,A -85,B 0,C 180,E1 -12301.249,E2 -12301.249} C_VEL
LIN {X 0,Y 376.12,Z 505.711,A -85,B 0,C 180,E1 -12304.547,E2 -12304.547} C_VEL
LIN {X 0,Y 375.603,Z 513.208,A -85,B 0,C 180,E1 -12308.023,E2 -12308.023} C_VEL
LIN {X 0,Y 375.374,Z 516.558,A -85,B 0,C 180,E1 -12309.557,E2 -12309.557} C_VEL
LIN {X 0,Y 378.867,Z 533.495,A -85,B 0,C 180,E1 -12310.716,E2 -12310.716} C_VEL
LIN {X 0,Y 380.022,Z 545.074,A -85,B 0,C 180,E1 -12311.586,E2 -12311.586} C_VEL
LIN {X 0,Y 380.49,Z 557.753,A -85,B 0,C 180,E1 -12312.672,E2 -12312.672} C_VEL
LIN {X 0,Y 379.282,Z 568.669,A -85,B 0,C 180,E1 -12313.724,E2 -12313.724} C_VEL
LIN {X 0,Y 378.028,Z 580.125,A -85,B 0,C 180,E1 -12315.088,E2 -12315.088} C_VEL
LIN {X 0,Y 376.99,Z 589.894,A -85,B 0,C 180,E1 -12316.524,E2 -12316.524} C_VEL
LIN {X 0,Y 376.035,Z 598.87,A -85,B 0,C 180,E1 -12318.136,E2 -12318.136} C_VEL
LIN {X 0,Y 375.368,Z 606.164,A -85,B 0,C 180,E1 -12319.754,E2 -12319.754} C_VEL
LIN {X 0,Y 374.97,Z 612.049,A -85,B 0,C 180,E1 -12321.376,E2 -12321.376} C_VEL
LIN {X 0,Y 374.75,Z 616.738,A -85,B 0,C 180,E1 -12322.998,E2 -12322.998} C_VEL
LIN {X 0,Y 374.613,Z 622.559,A -85,B 0,C 180,E1 -12325.696,E2 -12325.696} C_VEL
LIN {X 0,Y 374.598,Z 624.228,A -85,B 0,C 180,E1 -12326.773,E2 -12326.773} C_VEL
LIN {X 0,Y 374.711,Z 625.481,A -85,B 0,C 180,E1 -12327.85,E2 -12327.85} C_VEL
LIN {X 0,Y 374.67,Z 626.301,A -85,B 0,C 180,E1 -12328.925,E2 -12328.925} C_VEL
LIN {X 0,Y 374.665,Z 626.656,A -85,B 0,C 180,E1 -12330,E2 -12330} C_VEL
LIN {X 0,Y 374.663,Z 626.59,A -85,B 0,C 180,E1 -12331.075,E2 -12331.075} C_VEL
LIN {X 0,Y 374.67,Z 626.115,A -85,B 0,C 180,E1 -12332.15,E2 -12332.15} C_VEL
LIN {X 0,Y 374.553,Z 625.215,A -85,B 0,C 180,E1 -12333.227,E2 -12333.227} C_VEL
LIN {X 0,Y 374.585,Z 623.857,A -85,B 0,C 180,E1 -12334.304,E2 -12334.304} C_VEL
LIN {X 0,Y 374.589,Z 620.695,A -85,B 0,C 180,E1 -12336.077,E2 -12336.077} C_VEL
LIN {X 0,Y 374.875,Z 615.63,A -85,B 0,C 180,E1 -12338.083,E2 -12338.083} C_VEL
LIN {X 0,Y 375.332,Z 609.217,A -85,B 0,C 180,E1 -12339.974,E2 -12339.974} C_VEL
LIN {X 0,Y 375.969,Z 602.309,A -85,B 0,C 180,E1 -12341.593,E2 -12341.593} C_VEL
LIN {X 0,Y 376.843,Z 593.872,A -85,B 0,C 180,E1 -12343.206,E2 -12343.206} C_VEL
LIN {X 0,Y 377.803,Z 585.006,A -85,B 0,C 180,E1 -12344.602,E2 -12344.602} C_VEL
LIN {X 0,Y 379.291,Z 572.923,A -85,B 0,C 180,E1 -12346.137,E2 -12346.137} C_VEL
LIN {X 0,Y 380.681,Z 561.304,A -85,B 0,C 180,E1 -12347.319,E2 -12347.319} C_VEL
LIN {X 0,Y 380.996,Z 553.743,A -85,B 0,C 180,E1 -12347.998,E2 -12347.998} C_VEL
LIN {X 0,Y 380.44,Z 540.932,A -85,B 0,C 180,E1 -12349.031,E2 -12349.031} C_VEL
LIN {X 0,Y 378.629,Z 529.328,A -85,B 0,C 180,E1 -12349.893,E2 -12349.893} C_VEL
LIN {X 0,Y 375.481,Z 515.916,A -85,B 0,C 180,E1 -12350.832,E2 -12350.832} C_VEL
LIN {X 0,Y 375.961,Z 508.727,A -85,B 0,C 180,E1 -12354.284,E2 -12354.284} C_VEL
LIN {X 0,Y 376.65,Z 501.895,A -85,B 0,C 180,E1 -12357.806,E2 -12357.806} C_VEL
LIN {X 0,Y 377.435,Z 496.095,A -85,B 0,C 180,E1 -12361.07,E2 -12361.07} C_VEL
LIN {X 0,Y 378.208,Z 491.602,A -85,B 0,C 180,E1 -12363.881,E2 -12363.881} C_VEL
LIN {X 0,Y 378.723,Z 488.03,A -85,B 0,C 180,E1 -12366.429,E2 -12366.429} C_VEL
LIN {X 0,Y 378.673,Z 485.278,A -85,B 0,C 180,E1 -12368.785,E2 -12368.785} C_VEL
LIN {X 0,Y 378.209,Z 482.361,A -85,B 0,C 180,E1 -12371.987,E2 -12371.987} C_VEL
LIN {X 0,Y 377.868,Z 480.358,A -85,B 0,C 180,E1 -12375.028,E2 -12375.028} C_VEL
LIN {X 0,Y 377.607,Z 479.067,A -85,B 0,C 180,E1 -12378.115,E2 -12378.115} C_VEL
LIN {X 0,Y 377.403,Z 478.44,A -85,B 0,C 180,E1 -12381.456,E2 -12381.456} C_VEL
LIN {X 0,Y 377.324,Z 478.412,A -85,B 0,C 180,E1 -12383.414,E2 -12383.414} C_VEL
LIN {X 0,Y 376.941,Z 478.971,A -85,B 0,C 180,E1 -12387.037,E2 -12387.037} C_VEL
LIN {X 0,Y 376.6,Z 479.805,A -85,B 0,C 180,E1 -12389.744,E2 -12389.744} C_VEL
LIN {X 0,Y 376.155,Z 481.36,A -85,B 0,C 180,E1 -12393.358,E2 -12393.358} C_VEL
LIN {X 0,Y 375.855,Z 483.254,A -85,B 0,C 180,E1 -12396.879,E2 -12396.879} C_VEL
LIN {X 0,Y 375.739,Z 484.775,A -85,B 0,C 180,E1 -12399.359,E2 -12399.359} C_VEL
LIN {X 0,Y 376.815,Z 487.746,A -85,B 0,C 180,E1 -12399.611,E2 -12399.611} C_VEL
LIN {X 0,Y 380.882,Z 498.385,A -85,B 0,C 180,E1 -12400.602,E2 -12400.602} C_VEL
LIN {X 0,Y 383.589,Z 508.364,A -85,B 0,C 180,E1 -12401.534,E2 -12401.534} C_VEL
LIN {X 0,Y 382.652,Z 520.24,A -85,B 0,C 180,E1 -12402.497,E2 -12402.497} C_VEL
LIN {X 0,Y 381.433,Z 531.004,A -85,B 0,C 180,E1 -12403.578,E2 -12403.578} C_VEL
LIN {X 0,Y 380.039,Z 542.452,A -85,B 0,C 180,E1 -12404.995,E2 -12404.995} C_VEL
LIN {X 0,Y 378.881,Z 551.112,A -85,B 0,C 180,E1 -12406.32,E2 -12406.32} C_VEL
LIN {X 0,Y 377.797,Z 559.603,A -85,B 0,C 180,E1 -12407.92,E2 -12407.92} C_VEL
LIN {X 0,Y 376.933,Z 566.487,A -85,B 0,C 180,E1 -12409.526,E2 -12409.526} C_VEL
LIN {X 0,Y 376.363,Z 571.172,A -85,B 0,C 180,E1 -12410.867,E2 -12410.867} C_VEL
LIN {X 0,Y 375.72,Z 575.738,A -85,B 0,C 180,E1 -12412.476,E2 -12412.476} C_VEL
LIN {X 0,Y 375.359,Z 578.189,A -85,B 0,C 180,E1 -12413.55,E2 -12413.55} C_VEL
LIN {X 0,Y 375.232,Z 580.12,A -85,B 0,C 180,E1 -12414.627,E2 -12414.627} C_VEL
LIN {X 0,Y 375.15,Z 581.636,A -85,B 0,C 180,E1 -12415.703,E2 -12415.703} C_VEL
LIN {X 0,Y 374.958,Z 582.762,A -85,B 0,C 180,E1 -12416.777,E2 -12416.777} C_VEL
LIN {X 0,Y 374.828,Z 583.45,A -85,B 0,C 180,E1 -12417.851,E2 -12417.851} C_VEL
LIN {X 0,Y 374.723,Z 583.721,A -85,B 0,C 180,E1 -12418.926,E2 -12418.926} C_VEL
LIN {X 0,Y 374.667,Z 583.6,A -85,B 0,C 180,E1 -12420,E2 -12420} C_VEL
LIN {X 0,Y 374.679,Z 583.079,A -85,B 0,C 180,E1 -12421.075,E2 -12421.075} C_VEL
LIN {X 0,Y 374.772,Z 582.106,A -85,B 0,C 180,E1 -12422.15,E2 -12422.15} C_VEL
LIN {X 0,Y 374.792,Z 580.72,A -85,B 0,C 180,E1 -12423.225,E2 -12423.225} C_VEL
LIN {X 0,Y 374.866,Z 577.835,A -85,B 0,C 180,E1 -12424.84,E2 -12424.84} C_VEL
LIN {X 0,Y 375.106,Z 573.898,A -85,B 0,C 180,E1 -12426.455,E2 -12426.455} C_VEL
LIN {X 0,Y 375.368,Z 568.808,A -85,B 0,C 180,E1 -12428.073,E2 -12428.073} C_VEL
LIN {X 0,Y 375.865,Z 562.424,A -85,B 0,C 180,E1 -12429.688,E2 -12429.688} C_VEL
LIN {X 0,Y 376.448,Z 554.484,A -85,B 0,C 180,E1 -12431.305,E2 -12431.305} C_VEL
LIN {X 0,Y 377.218,Z 544.618,A -85,B 0,C 180,E1 -12432.919,E2 -12432.919} C_VEL
LIN {X 0,Y 378.065,Z 534.581,A -85,B 0,C 180,E1 -12434.247,E2 -12434.247} C_VEL
LIN {X 0,Y 378.819,Z 523.168,A -85,B 0,C 180,E1 -12435.467,E2 -12435.467} C_VEL
LIN {X 0,Y 379.627,Z 510.548,A -85,B 0,C 180,E1 -12436.537,E2 -12436.537} C_VEL
LIN {X 0,Y 379.981,Z 503.757,A -85,B 0,C 180,E1 -12437.006,E2 -12437.006} C_VEL
LIN {X 0,Y 377.511,Z 491.792,A -85,B 0,C 180,E1 -12437.785,E2 -12437.785} C_VEL
LIN {X 0,Y 374.848,Z 479.296,A -85,B 0,C 180,E1 -12438.429,E2 -12438.429} C_VEL
LIN {X 0,Y 374.847,Z 476.816,A -85,B 0,C 180,E1 -12440.869,E2 -12440.869} C_VEL
LIN {X 0,Y 374.937,Z 473.349,A -85,B 0,C 180,E1 -12444.355,E2 -12444.355} C_VEL
LIN {X 0,Y 375.115,Z 469.881,A -85,B 0,C 180,E1 -12447.93,E2 -12447.93} C_VEL
LIN {X 0,Y 375.444,Z 469.718,A -85,B 0,C 180,E1 -12451.611,E2 -12451.611} C_VEL
LIN {X 0,Y 375.847,Z 469.666,A -85,B 0,C 180,E1 -12455.428,E2 -12455.428} C_VEL
LIN {X 0,Y 375.973,Z 469.654,A -85,B 0,C 180,E1 -12458.27,E2 -12458.27} C_VEL
LIN {X 0,Y 375.939,Z 469.654,A -85,B 0,C 180,E1 -12461.601,E2 -12461.601} C_VEL
LIN {X 0,Y 375.932,Z 469.655,A -85,B 0,C 180,E1 -12465.269,E2 -12465.269} C_VEL
LIN {X 0,Y 375.939,Z 469.659,A -85,B 0,C 180,E1 -12468.399,E2 -12468.399} C_VEL
LIN {X 0,Y 375.98,Z 469.651,A -85,B 0,C 180,E1 -12471.729,E2 -12471.729} C_VEL
LIN {X 0,Y 375.984,Z 469.648,A -85,B 0,C 180,E1 -12475.333,E2 -12475.333} C_VEL
LIN {X 0,Y 375.962,Z 469.655,A -85,B 0,C 180,E1 -12478.438,E2 -12478.438} C_VEL
LIN {X 0,Y 376.001,Z 469.65,A -85,B 0,C 180,E1 -12482.142,E2 -12482.142} C_VEL
LIN {X 0,Y 376.011,Z 469.647,A -85,B 0,C 180,E1 -12484.539,E2 -12484.539} C_VEL
LIN {X 0,Y 375.968,Z 469.656,A -85,B 0,C 180,E1 -12488.046,E2 -12488.046} C_VEL
LIN {X 0,Y 376.028,Z 469.644,A -85,B 0,C 180,E1 -12491.474,E2 -12491.474} C_VEL
LIN {X 0,Y 376.064,Z 469.639,A -85,B 0,C 180,E1 -12494.833,E2 -12494.833} C_VEL
LIN {X 0,Y 376.055,Z 469.645,A -85,B 0,C 180,E1 -12498.137,E2 -12498.137} C_VEL
LIN {X 0,Y 376.263,Z 469.619,A -85,B 0,C 180,E1 -12501.877,E2 -12501.877} C_VEL
LIN {X 0,Y 376.176,Z 469.626,A -85,B 0,C 180,E1 -12504.64,E2 -12504.64} C_VEL
LIN {X 0,Y 376.357,Z 469.606,A -85,B 0,C 180,E1 -12507.86,E2 -12507.86} C_VEL
LIN {X 0,Y 376.493,Z 469.59,A -85,B 0,C 180,E1 -12510,E2 -12510} C_VEL
LIN {X 0,Y 376.189,Z 469.623,A -85,B 0,C 180,E1 -12513.213,E2 -12513.213} C_VEL
LIN {X 0,Y 376.219,Z 469.622,A -85,B 0,C 180,E1 -12516.435,E2 -12516.435} C_VEL
LIN {X 0,Y 376.118,Z 469.635,A -85,B 0,C 180,E1 -12519.682,E2 -12519.682} C_VEL
LIN {X 0,Y 376.094,Z 469.638,A -85,B 0,C 180,E1 -12523.658,E2 -12523.658} C_VEL
LIN {X 0,Y 376.049,Z 469.644,A -85,B 0,C 180,E1 -12527.607,E2 -12527.607} C_VEL
LIN {X 0,Y 375.983,Z 469.649,A -85,B 0,C 180,E1 -12530.832,E2 -12530.832} C_VEL
LIN {X 0,Y 375.994,Z 469.649,A -85,B 0,C 180,E1 -12534.282,E2 -12534.282} C_VEL
LIN {X 0,Y 376.024,Z 469.643,A -85,B 0,C 180,E1 -12536.652,E2 -12536.652} C_VEL
LIN {X 0,Y 375.969,Z 469.653,A -85,B 0,C 180,E1 -12540.312,E2 -12540.312} C_VEL
LIN {X 0,Y 375.967,Z 469.654,A -85,B 0,C 180,E1 -12544.111,E2 -12544.111} C_VEL
LIN {X 0,Y 375.95,Z 469.652,A -85,B 0,C 180,E1 -12546.029,E2 -12546.029} C_VEL
LIN {X 0,Y 375.303,Z 469.734,A -85,B 0,C 180,E1 -12546.923,E2 -12546.923} C_VEL
LIN {X 0,Y 372.468,Z 470.087,A -85,B 0,C 180,E1 -12548.377,E2 -12548.377} C_VEL
LIN {X 0,Y 370.043,Z 470.392,A -85,B 0,C 180,E1 -12549.553,E2 -12549.553} C_VEL
LIN {X 0,Y 368.981,Z 470.521,A -85,B 0,C 180,E1 -12550.462,E2 -12550.462} C_VEL
LIN {X 0,Y 368.884,Z 470.532,A -85,B 0,C 180,E1 -12550.77,E2 -12550.77} C_VEL
LIN {X 0,Y 368.887,Z 470.537,A -85,B 0,C 180,E1 -12553.616,E2 -12553.616} C_VEL
LIN {X 0,Y 368.89,Z 470.532,A -85,B 0,C 180,E1 -12556.696,E2 -12556.696} C_VEL
LIN {X 0,Y 368.916,Z 470.533,A -85,B 0,C 180,E1 -12559.643,E2 -12559.643} C_VEL
LIN {X 0,Y 368.887,Z 470.533,A -85,B 0,C 180,E1 -12563.148,E2 -12563.148} C_VEL
LIN {X 0,Y 368.689,Z 470.558,A -85,B 0,C 180,E1 -12566.44,E2 -12566.44} C_VEL
LIN {X 0,Y 368.389,Z 470.597,A -85,B 0,C 180,E1 -12569.148,E2 -12569.148} C_VEL
LIN {X 0,Y 367.959,Z 470.653,A -85,B 0,C 180,E1 -12572.716,E2 -12572.716} C_VEL
LIN {X 0,Y 367.847,Z 470.892,A -85,B 0,C 180,E1 -12573.932,E2 -12573.932} C_VEL
LIN {X 0,Y 367.729,Z 474.825,A -85,B 0,C 180,E1 -12577.527,E2 -12577.527} C_VEL
LIN {X 0,Y 367.752,Z 477.396,A -85,B 0,C 180,E1 -12579.879,E2 -12579.879} C_VEL
LIN {X 0,Y 367.737,Z 479.138,A -85,B 0,C 180,E1 -12581.438,E2 -12581.438} C_VEL
LIN {X 0,Y 370.822,Z 494.132,A -85,B 0,C 180,E1 -12582.244,E2 -12582.244} C_VEL
LIN {X 0,Y 372.917,Z 504.41,A -85,B 0,C 180,E1 -12582.945,E2 -12582.945} C_VEL
LIN {X 0,Y 372.192,Z 517.787,A -85,B 0,C 180,E1 -12583.968,E2 -12583.968} C_VEL
LIN {X 0,Y 371.509,Z 528.838,A -85,B 0,C 180,E1 -12585.05,E2 -12585.05} C_VEL
LIN {X 0,Y 370.556,Z 540.201,A -85,B 0,C 180,E1 -12586.425,E2 -12586.425} C_VEL
LIN {X 0,Y 369.695,Z 550.175,A -85,B 0,C 180,E1 -12587.929,E2 -12587.929} C_VEL
LIN {X 0,Y 369.036,Z 559.014,A -85,B 0,C 180,E1 -12589.576,E2 -12589.576} C_VEL
LIN {X 0,Y 368.48,Z 566.117,A -85,B 0,C 180,E1 -12591.223,E2 -12591.223} C_VEL
LIN {X 0,Y 368.067,Z 572.721,A -85,B 0,C 180,E1 -12593.173,E2 -12593.173} C_VEL
LIN {X 0,Y 367.801,Z 577.537,A -85,B 0,C 180,E1 -12595.067,E2 -12595.067} C_VEL
LIN {X 0,Y 367.694,Z 580.558,A -85,B 0,C 180,E1 -12596.713,E2 -12596.713} C_VEL
LIN {X 0,Y 367.684,Z 582.004,A -85,B 0,C 180,E1 -12597.809,E2 -12597.809} C_VEL
LIN {X 0,Y 367.604,Z 583.054,A -85,B 0,C 180,E1 -12598.904,E2 -12598.904} C_VEL
LIN {X 0,Y 367.587,Z 583.696,A -85,B 0,C 180,E1 -12600,E2 -12600} C_VEL
LIN {X 0,Y 367.635,Z 583.883,A -85,B 0,C 180,E1 -12601.095,E2 -12601.095} C_VEL
LIN {X 0,Y 367.752,Z 583.672,A -85,B 0,C 180,E1 -12602.19,E2 -12602.19} C_VEL
LIN {X 0,Y 367.908,Z 583.07,A -85,B 0,C 180,E1 -12603.285,E2 -12603.285} C_VEL
LIN {X 0,Y 368.088,Z 582.023,A -85,B 0,C 180,E1 -12604.38,E2 -12604.38} C_VEL
LIN {X 0,Y 368.094,Z 580.573,A -85,B 0,C 180,E1 -12605.478,E2 -12605.478} C_VEL
LIN {X 0,Y 368.512,Z 577.756,A -85,B 0,C 180,E1 -12607.028,E2 -12607.028} C_VEL
LIN {X 0,Y 369.063,Z 573.532,A -85,B 0,C 180,E1 -12608.762,E2 -12608.762} C_VEL
LIN {X 0,Y 369.794,Z 568.345,A -85,B 0,C 180,E1 -12610.402,E2 -12610.402} C_VEL
LIN {X 0,Y 370.652,Z 561.875,A -85,B 0,C 180,E1 -12612.039,E2 -12612.039} C_VEL
LIN {X 0,Y 371.83,Z 553.789,A -85,B 0,C 180,E1 -12613.666,E2 -12613.666} C_VEL
LIN {X 0,Y 372.701,Z 547.452,A -85,B 0,C 180,E1 -12614.748,E2 -12614.748} C_VEL
LIN {X 0,Y 374.003,Z 538.002,A -85,B 0,C 180,E1 -12616.091,E2 -12616.091} C_VEL
LIN {X 0,Y 375.195,Z 527.949,A -85,B 0,C 180,E1 -12617.274,E2 -12617.274} C_VEL
LIN {X 0,Y 376.53,Z 516.433,A -85,B 0,C 180,E1 -12618.359,E2 -12618.359} C_VEL
LIN {X 0,Y 377.007,Z 509.663,A -85,B 0,C 180,E1 -12618.909,E2 -12618.909} C_VEL
LIN {X 0,Y 374.593,Z 499.774,A -85,B 0,C 180,E1 -12619.876,E2 -12619.876} C_VEL
LIN {X 0,Y 370.974,Z 489.895,A -85,B 0,C 180,E1 -12620.83,E2 -12620.83} C_VEL
LIN {X 0,Y 368.611,Z 484.011,A -85,B 0,C 180,E1 -12621.385,E2 -12621.385} C_VEL
LIN {X 0,Y 368.743,Z 480.524,A -85,B 0,C 180,E1 -12624.791,E2 -12624.791} C_VEL
LIN {X 0,Y 368.805,Z 478.176,A -85,B 0,C 180,E1 -12627.216,E2 -12627.216} C_VEL
LIN {X 0,Y 368.928,Z 475.792,A -85,B 0,C 180,E1 -12629.689,E2 -12629.689} C_VEL
LIN {X 0,Y 369.008,Z 472.623,A -85,B 0,C 180,E1 -12633.069,E2 -12633.069} C_VEL
LIN {X 0,Y 368.853,Z 470.54,A -85,B 0,C 180,E1 -12635.536,E2 -12635.536} C_VEL
LIN {X 0,Y 368.905,Z 470.533,A -85,B 0,C 180,E1 -12638.953,E2 -12638.953} C_VEL
LIN {X 0,Y 368.884,Z 470.535,A -85,B 0,C 180,E1 -12642.009,E2 -12642.009} C_VEL
LIN {X 0,Y 368.961,Z 470.594,A -85,B 0,C 180,E1 -12645.884,E2 -12645.884} C_VEL
LIN {X 0,Y 370.036,Z 476.663,A -85,B 0,C 180,E1 -12649.439,E2 -12649.439} C_VEL
LIN {X 0,Y 371.015,Z 482.539,A -85,B 0,C 180,E1 -12652.711,E2 -12652.711} C_VEL
LIN {X 0,Y 371.089,Z 485.97,A -85,B 0,C 180,E1 -12654.525,E2 -12654.525} C_VEL
LIN {X 0,Y 370.36,Z 492.649,A -85,B 0,C 180,E1 -12657.904,E2 -12657.904} C_VEL
LIN {X 0,Y 369.625,Z 500.198,A -85,B 0,C 180,E1 -12661.618,E2 -12661.618} C_VEL
LIN {X 0,Y 368.947,Z 507.693,A -85,B 0,C 180,E1 -12665.224,E2 -12665.224} C_VEL
LIN {X 0,Y 368.387,Z 515.474,A -85,B 0,C 180,E1 -12668.891,E2 -12668.891} C_VEL
LIN {X 0,Y 369.183,Z 519.243,A -85,B 0,C 180,E1 -12669.133,E2 -12669.133} C_VEL
LIN {X 0,Y 371.868,Z 531.596,A -85,B 0,C 180,E1 -12670.04,E2 -12670.04} C_VEL
LIN {X 0,Y 373.23,Z 541.863,A -85,B 0,C 180,E1 -12670.843,E2 -12670.843} C_VEL
LIN {X 0,Y 373.824,Z 555.958,A -85,B 0,C 180,E1 -12672.07,E2 -12672.07} C_VEL
LIN {X 0,Y 373.459,Z 561.729,A -85,B 0,C 180,E1 -12672.618,E2 -12672.618} C_VEL
LIN {X 0,Y 372.105,Z 572.942,A -85,B 0,C 180,E1 -12673.824,E2 -12673.824} C_VEL
LIN {X 0,Y 370.848,Z 583.545,A -85,B 0,C 180,E1 -12675.22,E2 -12675.22} C_VEL
LIN {X 0,Y 369.714,Z 593.304,A -85,B 0,C 180,E1 -12676.814,E2 -12676.814} C_VEL
LIN {X 0,Y 368.82,Z 601.521,A -85,B 0,C 180,E1 -12678.458,E2 -12678.458} C_VEL
LIN {X 0,Y 368.17,Z 608.244,A -85,B 0,C 180,E1 -12680.107,E2 -12680.107} C_VEL
LIN {X 0,Y 367.821,Z 613.625,A -85,B 0,C 180,E1 -12681.761,E2 -12681.761} C_VEL
LIN {X 0,Y 367.6,Z 618.667,A -85,B 0,C 180,E1 -12683.81,E2 -12683.81} C_VEL
LIN {X 0,Y 367.55,Z 621.945,A -85,B 0,C 180,E1 -12685.613,E2 -12685.613} C_VEL
LIN {X 0,Y 367.511,Z 623.653,A -85,B 0,C 180,E1 -12686.711,E2 -12686.711} C_VEL
LIN {X 0,Y 367.644,Z 624.937,A -85,B 0,C 180,E1 -12687.809,E2 -12687.809} C_VEL
LIN {X 0,Y 367.604,Z 625.79,A -85,B 0,C 180,E1 -12688.905,E2 -12688.905} C_VEL
LIN {X 0,Y 367.595,Z 626.204,A -85,B 0,C 180,E1 -12690,E2 -12690} C_VEL
LIN {X 0,Y 367.596,Z 626.166,A -85,B 0,C 180,E1 -12691.096,E2 -12691.096} C_VEL
LIN {X 0,Y 367.57,Z 625.717,A -85,B 0,C 180,E1 -12692.192,E2 -12692.192} C_VEL
LIN {X 0,Y 367.465,Z 624.855,A -85,B 0,C 180,E1 -12693.289,E2 -12693.289} C_VEL
LIN {X 0,Y 367.51,Z 623.551,A -85,B 0,C 180,E1 -12694.387,E2 -12694.387} C_VEL
LIN {X 0,Y 367.489,Z 620.796,A -85,B 0,C 180,E1 -12696.029,E2 -12696.029} C_VEL
LIN {X 0,Y 367.705,Z 616.983,A -85,B 0,C 180,E1 -12697.689,E2 -12697.689} C_VEL
LIN {X 0,Y 368.064,Z 612.074,A -85,B 0,C 180,E1 -12699.341,E2 -12699.341} C_VEL
LIN {X 0,Y 368.7,Z 604.787,A -85,B 0,C 180,E1 -12701.267,E2 -12701.267} C_VEL
LIN {X 0,Y 369.627,Z 597.024,A -85,B 0,C 180,E1 -12702.91,E2 -12702.91} C_VEL
LIN {X 0,Y 370.561,Z 588.215,A -85,B 0,C 180,E1 -12704.446,E2 -12704.446} C_VEL
LIN {X 0,Y 372.086,Z 576.887,A -85,B 0,C 180,E1 -12706.036,E2 -12706.036} C_VEL
LIN {X 0,Y 373.448,Z 566.353,A -85,B 0,C 180,E1 -12707.242,E2 -12707.242} C_VEL
LIN {X 0,Y 374.386,Z 556.572,A -85,B 0,C 180,E1 -12708.185,E2 -12708.185} C_VEL
LIN {X 0,Y 373.989,Z 542.868,A -85,B 0,C 180,E1 -12709.373,E2 -12709.373} C_VEL
LIN {X 0,Y 372.444,Z 531.854,A -85,B 0,C 180,E1 -12710.26,E2 -12710.26} C_VEL
LIN {X 0,Y 369.579,Z 519.287,A -85,B 0,C 180,E1 -12711.204,E2 -12711.204} C_VEL
LIN {X 0,Y 368.494,Z 515.265,A -85,B 0,C 180,E1 -12711.51,E2 -12711.51} C_VEL
LIN {X 0,Y 369.03,Z 508.719,A -85,B 0,C 180,E1 -12714.77,E2 -12714.77} C_VEL
LIN {X 0,Y 369.743,Z 501.988,A -85,B 0,C 180,E1 -12718.372,E2 -12718.372} C_VEL
LIN {X 0,Y 370.508,Z 496.819,A -85,B 0,C 180,E1 -12721.396,E2 -12721.396} C_VEL
LIN {X 0,Y 371.394,Z 491.942,A -85,B 0,C 180,E1 -12724.59,E2 -12724.59} C_VEL
LIN {X 0,Y 371.822,Z 488.234,A -85,B 0,C 180,E1 -12727.452,E2 -12727.452} C_VEL
LIN {X 0,Y 371.525,Z 485.574,A -85,B 0,C 180,E1 -12730.028,E2 -12730.028} C_VEL
LIN {X 0,Y 371.13,Z 483.194,A -85,B 0,C 180,E1 -12732.979,E2 -12732.979} C_VEL
LIN {X 0,Y 370.85,Z 481.403,A -85,B 0,C 180,E1 -12736.066,E2 -12736.066} C_VEL
LIN {X 0,Y 370.57,Z 480.292,A -85,B 0,C 180,E1 -12739.343,E2 -12739.343} C_VEL
LIN {X 0,Y 370.378,Z 479.888,A -85,B 0,C 180,E1 -12742.841,E2 -12742.841} C_VEL
LIN {X 0,Y 370.145,Z 480.056,A -85,B 0,C 180,E1 -12745.277,E2 -12745.277} C_VEL
LIN {X 0,Y 369.86,Z 480.573,A -85,B 0,C 180,E1 -12747.856,E2 -12747.856} C_VEL
LIN {X 0,Y 369.458,Z 481.63,A -85,B 0,C 180,E1 -12751.049,E2 -12751.049} C_VEL
LIN {X 0,Y 369.117,Z 482.938,A -85,B 0,C 180,E1 -12754.029,E2 -12754.029} C_VEL
LIN {X 0,Y 368.794,Z 484.855,A -85,B 0,C 180,E1 -12757.596,E2 -12757.596} C_VEL
LIN {X 0,Y 368.714,Z 485.491,A -85,B 0,C 180,E1 -12758.676,E2 -12758.676} C_VEL
LIN {X 0,Y 369.991,Z 488.744,A -85,B 0,C 180,E1 -12758.987,E2 -12758.987} C_VEL
LIN {X 0,Y 373.997,Z 498.661,A -85,B 0,C 180,E1 -12759.982,E2 -12759.982} C_VEL
LIN {X 0,Y 377.184,Z 510.069,A -85,B 0,C 180,E1 -12761.13,E2 -12761.13} C_VEL
LIN {X 0,Y 376.087,Z 522.383,A -85,B 0,C 180,E1 -12762.182,E2 -12762.182} C_VEL
LIN {X 0,Y 374.677,Z 534.133,A -85,B 0,C 180,E1 -12763.428,E2 -12763.428} C_VEL
LIN {X 0,Y 373.356,Z 543.944,A -85,B 0,C 180,E1 -12764.72,E2 -12764.72} C_VEL
LIN {X 0,Y 372.095,Z 552.365,A -85,B 0,C 180,E1 -12766.065,E2 -12766.065} C_VEL
LIN {X 0,Y 370.961,Z 560.727,A -85,B 0,C 180,E1 -12767.694,E2 -12767.694} C_VEL
LIN {X 0,Y 370.025,Z 567.5,A -85,B 0,C 180,E1 -12769.328,E2 -12769.328} C_VEL
LIN {X 0,Y 369.417,Z 572.075,A -85,B 0,C 180,E1 -12770.694,E2 -12770.694} C_VEL
LIN {X 0,Y 368.722,Z 576.609,A -85,B 0,C 180,E1 -12772.37,E2 -12772.37} C_VEL
LIN {X 0,Y 368.345,Z 578.883,A -85,B 0,C 180,E1 -12773.427,E2 -12773.427} C_VEL
LIN {X 0,Y 368.183,Z 580.776,A -85,B 0,C 180,E1 -12774.523,E2 -12774.523} C_VEL
LIN {X 0,Y 368.111,Z 582.252,A -85,B 0,C 180,E1 -12775.62,E2 -12775.62} C_VEL
LIN {X 0,Y 367.91,Z 583.329,A -85,B 0,C 180,E1 -12776.715,E2 -12776.715} C_VEL
LIN {X 0,Y 367.766,Z 583.956,A -85,B 0,C 180,E1 -12777.81,E2 -12777.81} C_VEL
LIN {X 0,Y 367.655,Z 584.188,A -85,B 0,C 180,E1 -12778.905,E2 -12778.905} C_VEL
LIN {X 0,Y 367.598,Z 584.023,A -85,B 0,C 180,E1 -12780,E2 -12780} C_VEL
LIN {X 0,Y 367.613,Z 583.438,A -85,B 0,C 180,E1 -12781.096,E2 -12781.096} C_VEL
LIN {X 0,Y 367.691,Z 582.412,A -85,B 0,C 180,E1 -12782.191,E2 -12782.191} C_VEL
LIN {X 0,Y 367.7,Z 580.99,A -85,B 0,C 180,E1 -12783.287,E2 -12783.287} C_VEL
LIN {X 0,Y 367.809,Z 578.03,A -85,B 0,C 180,E1 -12784.933,E2 -12784.933} C_VEL
LIN {X 0,Y 368.059,Z 574.011,A -85,B 0,C 180,E1 -12786.579,E2 -12786.579} C_VEL
LIN {X 0,Y 368.407,Z 567.853,A -85,B 0,C 180,E1 -12788.502,E2 -12788.502} C_VEL
LIN {X 0,Y 368.925,Z 561.089,A -85,B 0,C 180,E1 -12790.15,E2 -12790.15} C_VEL
LIN {X 0,Y 369.563,Z 552.733,A -85,B 0,C 180,E1 -12791.797,E2 -12791.797} C_VEL
LIN {X 0,Y 370.265,Z 544.25,A -85,B 0,C 180,E1 -12793.166,E2 -12793.166} C_VEL
LIN {X 0,Y 371.117,Z 534.253,A -85,B 0,C 180,E1 -12794.488,E2 -12794.488} C_VEL
LIN {X 0,Y 371.916,Z 522.386,A -85,B 0,C 180,E1 -12795.762,E2 -12795.762} C_VEL
LIN {X 0,Y 372.644,Z 511.251,A -85,B 0,C 180,E1 -12796.715,E2 -12796.715} C_VEL
LIN {X 0,Y 373.016,Z 504.512,A -85,B 0,C 180,E1 -12797.192,E2 -12797.192} C_VEL
LIN {X 0,Y 370.157,Z 490.853,A -85,B 0,C 180,E1 -12798.1,E2 -12798.1} C_VEL
LIN {X 0,Y 367.789,Z 479.665,A -85,B 0,C 180,E1 -12798.667,E2 -12798.667} C_VEL
LIN {X 0,Y 367.766,Z 477.026,A -85,B 0,C 180,E1 -12801.29,E2 -12801.29} C_VEL
LIN {X 0,Y 367.907,Z 473.52,A -85,B 0,C 180,E1 -12804.851,E2 -12804.851} C_VEL
LIN {X 0,Y 367.977,Z 471.181,A -85,B 0,C 180,E1 -12807.283,E2 -12807.283} C_VEL
LIN {X 0,Y 368.12,Z 470.637,A -85,B 0,C 180,E1 -12808.572,E2 -12808.572} C_VEL
LIN {X 0,Y 368.466,Z 470.59,A -85,B 0,C 180,E1 -12812.281,E2 -12812.281} C_VEL
LIN {X 0,Y 368.764,Z 470.549,A -85,B 0,C 180,E1 -12814.964,E2 -12814.964} C_VEL
LIN {X 0,Y 368.877,Z 470.534,A -85,B 0,C 180,E1 -12817.567,E2 -12817.567} C_VEL
LIN {X 0,Y 368.914,Z 470.534,A -85,B 0,C 180,E1 -12820.37,E2 -12820.37} C_VEL
LIN {X 0,Y 368.887,Z 470.533,A -85,B 0,C 180,E1 -12823.616,E2 -12823.616} C_VEL
LIN {X 0,Y 368.89,Z 470.535,A -85,B 0,C 180,E1 -12826.696,E2 -12826.696} C_VEL
LIN {X 0,Y 368.916,Z 470.53,A -85,B 0,C 180,E1 -12829.643,E2 -12829.643} C_VEL
LIN {X 0,Y 368.907,Z 470.529,A -85,B 0,C 180,E1 -12833.144,E2 -12833.144} C_VEL
LIN {X 0,Y 368.902,Z 470.534,A -85,B 0,C 180,E1 -12836.462,E2 -12836.462} C_VEL
LIN {X 0,Y 368.933,Z 470.527,A -85,B 0,C 180,E1 -12839.047,E2 -12839.047} C_VEL
LIN {X 0,Y 368.984,Z 470.522,A -85,B 0,C 180,E1 -12841.564,E2 -12841.564} C_VEL
LIN {X 0,Y 369.004,Z 470.522,A -85,B 0,C 180,E1 -12844.02,E2 -12844.02} C_VEL
LIN {X 0,Y 368.937,Z 470.527,A -85,B 0,C 180,E1 -12847.605,E2 -12847.605} C_VEL
LIN {X 0,Y 368.987,Z 470.52,A -85,B 0,C 180,E1 -12851.107,E2 -12851.107} C_VEL
LIN {X 0,Y 369.003,Z 470.52,A -85,B 0,C 180,E1 -12854.535,E2 -12854.535} C_VEL
LIN {X 0,Y 369.011,Z 470.521,A -85,B 0,C 180,E1 -12857.907,E2 -12857.907} C_VEL
LIN {X 0,Y 369.235,Z 470.493,A -85,B 0,C 180,E1 -12861.8,E2 -12861.8} C_VEL
LIN {X 0,Y 369.149,Z 470.502,A -85,B 0,C 180,E1 -12864.538,E2 -12864.538} C_VEL
LIN {X 0,Y 369.322,Z 470.482,A -85,B 0,C 180,E1 -12867.819,E2 -12867.819} C_VEL
LIN {X 0,Y 369.462,Z 470.466,A -85,B 0,C 180,E1 -12870,E2 -12870} C_VEL
LIN {X 0,Y 369.322,Z 470.482,A -85,B 0,C 180,E1 -12872.181,E2 -12872.181} C_VEL
LIN {X 0,Y 369.178,Z 470.498,A -85,B 0,C 180,E1 -12876.559,E2 -12876.559} C_VEL
LIN {X 0,Y 369.068,Z 470.514,A -85,B 0,C 180,E1 -12879.868,E2 -12879.868} C_VEL
LIN {X 0,Y 369.042,Z 470.517,A -85,B 0,C 180,E1 -12883.772,E2 -12883.772} C_VEL
LIN {X 0,Y 369.006,Z 470.523,A -85,B 0,C 180,E1 -12887.768,E2 -12887.768} C_VEL
LIN {X 0,Y 368.914,Z 470.53,A -85,B 0,C 180,E1 -12891.221,E2 -12891.221} C_VEL
LIN {X 0,Y 368.96,Z 470.523,A -85,B 0,C 180,E1 -12894.775,E2 -12894.775} C_VEL
LIN {X 0,Y 368.968,Z 470.523,A -85,B 0,C 180,E1 -12897.203,E2 -12897.203} C_VEL
LIN {X 0,Y 368.933,Z 470.527,A -85,B 0,C 180,E1 -12900.953,E2 -12900.953} C_VEL
LIN {X 0,Y 368.934,Z 470.527,A -85,B 0,C 180,E1 -12905.001,E2 -12905.001} C_VEL
LIN {X 0,Y 368.914,Z 470.528,A -85,B 0,C 180,E1 -12908.64,E2 -12908.64} C_VEL
LIN {X 0,Y 368.884,Z 470.532,A -85,B 0,C 180,E1 -12910.77,E2 -12910.77} C_VEL
LIN {X 0,Y 368.178,Z 470.626,A -85,B 0,C 180,E1 -12911.682,E2 -12911.682} C_VEL
LIN {X 0,Y 365.285,Z 470.982,A -85,B 0,C 180,E1 -12913.163,E2 -12913.163} C_VEL
LIN {X 0,Y 362.878,Z 471.282,A -85,B 0,C 180,E1 -12914.361,E2 -12914.361} C_VEL
LIN {X 0,Y 361.883,Z 471.407,A -85,B 0,C 180,E1 -12915.288,E2 -12915.288} C_VEL
LIN {X 0,Y 361.821,Z 471.417,A -85,B 0,C 180,E1 -12915.602,E2 -12915.602} C_VEL
LIN {X 0,Y 361.84,Z 471.412,A -85,B 0,C 180,E1 -12919.244,E2 -12919.244} C_VEL
LIN {X 0,Y 361.855,Z 471.408,A -85,B 0,C 180,E1 -12922.779,E2 -12922.779} C_VEL
LIN {X 0,Y 361.708,Z 471.432,A -85,B 0,C 180,E1 -12925.703,E2 -12925.703} C_VEL
LIN {X 0,Y 361.368,Z 471.47,A -85,B 0,C 180,E1 -12928.84,E2 -12928.84} C_VEL
LIN {X 0,Y 360.98,Z 471.523,A -85,B 0,C 180,E1 -12932.143,E2 -12932.143} C_VEL
LIN {X 0,Y 360.802,Z 471.547,A -85,B 0,C 180,E1 -12933.641,E2 -12933.641} C_VEL
LIN {X 0,Y 360.665,Z 473.61,A -85,B 0,C 180,E1 -12935.844,E2 -12935.844} C_VEL
LIN {X 0,Y 360.692,Z 477.576,A -85,B 0,C 180,E1 -12939.468,E2 -12939.468} C_VEL
LIN {X 0,Y 360.673,Z 479.501,A -85,B 0,C 180,E1 -12941.213,E2 -12941.213} C_VEL
LIN {X 0,Y 363.336,Z 492.599,A -85,B 0,C 180,E1 -12941.891,E2 -12941.891} C_VEL
LIN {X 0,Y 365.866,Z 504.925,A -85,B 0,C 180,E1 -12942.735,E2 -12942.735} C_VEL
LIN {X 0,Y 365.301,Z 516.809,A -85,B 0,C 180,E1 -12943.658,E2 -12943.658} C_VEL
LIN {X 0,Y 364.625,Z 527.522,A -85,B 0,C 180,E1 -12944.691,E2 -12944.691} C_VEL
LIN {X 0,Y 363.715,Z 538.651,A -85,B 0,C 180,E1 -12946.022,E2 -12946.022} C_VEL
LIN {X 0,Y 362.872,Z 548.142,A -85,B 0,C 180,E1 -12947.415,E2 -12947.415} C_VEL
LIN {X 0,Y 362.237,Z 556.028,A -85,B 0,C 180,E1 -12948.812,E2 -12948.812} C_VEL
LIN {X 0,Y 361.625,Z 563.775,A -85,B 0,C 180,E1 -12950.491,E2 -12950.491} C_VEL
LIN {X 0,Y 361.161,Z 570.014,A -85,B 0,C 180,E1 -12952.171,E2 -12952.171} C_VEL
LIN {X 0,Y 360.862,Z 575.377,A -85,B 0,C 180,E1 -12954.001,E2 -12954.001} C_VEL
LIN {X 0,Y 360.659,Z 578.802,A -85,B 0,C 180,E1 -12955.529,E2 -12955.529} C_VEL
LIN {X 0,Y 360.601,Z 580.79,A -85,B 0,C 180,E1 -12956.648,E2 -12956.648} C_VEL
LIN {X 0,Y 360.605,Z 582.287,A -85,B 0,C 180,E1 -12957.766,E2 -12957.766} C_VEL
LIN {X 0,Y 360.54,Z 583.382,A -85,B 0,C 180,E1 -12958.883,E2 -12958.883} C_VEL
LIN {X 0,Y 360.52,Z 584.081,A -85,B 0,C 180,E1 -12960,E2 -12960} C_VEL
LIN {X 0,Y 360.57,Z 584.332,A -85,B 0,C 180,E1 -12961.117,E2 -12961.117} C_VEL
LIN {X 0,Y 360.693,Z 584.161,A -85,B 0,C 180,E1 -12962.233,E2 -12962.233} C_VEL
LIN {X 0,Y 360.861,Z 583.597,A -85,B 0,C 180,E1 -12963.349,E2 -12963.349} C_VEL
LIN {X 0,Y 361.046,Z 582.631,A -85,B 0,C 180,E1 -12964.465,E2 -12964.465} C_VEL
LIN {X 0,Y 361.052,Z 581.237,A -85,B 0,C 180,E1 -12965.585,E2 -12965.585} C_VEL
LIN {X 0,Y 361.721,Z 577.334,A -85,B 0,C 180,E1 -12967.735,E2 -12967.735} C_VEL
LIN {X 0,Y 362.373,Z 572.838,A -85,B 0,C 180,E1 -12969.488,E2 -12969.488} C_VEL
LIN {X 0,Y 363.383,Z 566.266,A -85,B 0,C 180,E1 -12971.434,E2 -12971.434} C_VEL
LIN {X 0,Y 364.391,Z 559.263,A -85,B 0,C 180,E1 -12973.098,E2 -12973.098} C_VEL
LIN {X 0,Y 365.672,Z 550.543,A -85,B 0,C 180,E1 -12974.753,E2 -12974.753} C_VEL
LIN {X 0,Y 367.047,Z 541.662,A -85,B 0,C 180,E1 -12976.119,E2 -12976.119} C_VEL
LIN {X 0,Y 368.594,Z 530.125,A -85,B 0,C 180,E1 -12977.568,E2 -12977.568} C_VEL
LIN {X 0,Y 370.064,Z 518.932,A -85,B 0,C 180,E1 -12978.692,E2 -12978.692} C_VEL
LIN {X 0,Y 370.67,Z 511.467,A -85,B 0,C 180,E1 -12979.334,E2 -12979.334} C_VEL
LIN {X 0,Y 368.036,Z 500.847,A -85,B 0,C 180,E1 -12980.429,E2 -12980.429} C_VEL
LIN {X 0,Y 364.125,Z 490.59,A -85,B 0,C 180,E1 -12981.513,E2 -12981.513} C_VEL
LIN {X 0,Y 361.66,Z 484.524,A -85,B 0,C 180,E1 -12982.14,E2 -12982.14} C_VEL
LIN {X 0,Y 361.817,Z 481.488,A -85,B 0,C 180,E1 -12985.298,E2 -12985.298} C_VEL
LIN {X 0,Y 361.97,Z 477.916,A -85,B 0,C 180,E1 -12989.106,E2 -12989.106} C_VEL
LIN {X 0,Y 362.085,Z 475.661,A -85,B 0,C 180,E1 -12991.605,E2 -12991.605} C_VEL
LIN {X 0,Y 362.047,Z 473.39,A -85,B 0,C 180,E1 -12994.26,E2 -12994.26} C_VEL
LIN {X 0,Y 361.856,Z 471.413,A -85,B 0,C 180,E1 -12997.019,E2 -12997.019} C_VEL
LIN {X 0,Y 361.857,Z 471.412,A -85,B 0,C 180,E1 -12999.861,E2 -12999.861} C_VEL
LIN {X 0,Y 361.838,Z 471.413,A -85,B 0,C 180,E1 -13002.829,E2 -13002.829} C_VEL
LIN {X 0,Y 361.906,Z 471.46,A -85,B 0,C 180,E1 -13005.645,E2 -13005.645} C_VEL
LIN {X 0,Y 362.91,Z 477.142,A -85,B 0,C 180,E1 -13009.048,E2 -13009.048} C_VEL
LIN {X 0,Y 363.908,Z 482.936,A -85,B 0,C 180,E1 -13012.355,E2 -13012.355} C_VEL
LIN {X 0,Y 364.099,Z 486.26,A -85,B 0,C 180,E1 -13014.165,E2 -13014.165} C_VEL
LIN {X 0,Y 363.592,Z 491.145,A -85,B 0,C 180,E1 -13016.707,E2 -13016.707} C_VEL
LIN {X 0,Y 362.747,Z 498.975,A -85,B 0,C 180,E1 -13020.674,E2 -13020.674} C_VEL
LIN {X 0,Y 362.035,Z 505.908,A -85,B 0,C 180,E1 -13024.101,E2 -13024.101} C_VEL
LIN {X 0,Y 361.427,Z 513.965,A -85,B 0,C 180,E1 -13028.018,E2 -13028.018} C_VEL
LIN {X 0,Y 361.418,Z 514.227,A -85,B 0,C 180,E1 -13028.13,E2 -13028.13} C_VEL
LIN {X 0,Y 362.146,Z 517.876,A -85,B 0,C 180,E1 -13028.379,E2 -13028.379} C_VEL
LIN {X 0,Y 365.018,Z 530.334,A -85,B 0,C 180,E1 -13029.362,E2 -13029.362} C_VEL
LIN {X 0,Y 366.741,Z 542.55,A -85,B 0,C 180,E1 -13030.379,E2 -13030.379} C_VEL
LIN {X 0,Y 367.174,Z 555.849,A -85,B 0,C 180,E1 -13031.589,E2 -13031.589} C_VEL
LIN {X 0,Y 367.139,Z 560.11,A -85,B 0,C 180,E1 -13032.021,E2 -13032.021} C_VEL
LIN {X 0,Y 365.784,Z 570.368,A -85,B 0,C 180,E1 -13033.106,E2 -13033.106} C_VEL
LIN {X 0,Y 364.334,Z 581.566,A -85,B 0,C 180,E1 -13034.576,E2 -13034.576} C_VEL
LIN {X 0,Y 363.204,Z 590.525,A -85,B 0,C 180,E1 -13036.003,E2 -13036.003} C_VEL
LIN {X 0,Y 362.144,Z 599.143,A -85,B 0,C 180,E1 -13037.674,E2 -13037.674} C_VEL
LIN {X 0,Y 361.35,Z 606.156,A -85,B 0,C 180,E1 -13039.352,E2 -13039.352} C_VEL
LIN {X 0,Y 360.863,Z 611.853,A -85,B 0,C 180,E1 -13041.037,E2 -13041.037} C_VEL
LIN {X 0,Y 360.594,Z 616.37,A -85,B 0,C 180,E1 -13042.722,E2 -13042.722} C_VEL
LIN {X 0,Y 360.484,Z 619.793,A -85,B 0,C 180,E1 -13044.406,E2 -13044.406} C_VEL
LIN {X 0,Y 360.426,Z 623.065,A -85,B 0,C 180,E1 -13046.646,E2 -13046.646} C_VEL
LIN {X 0,Y 360.559,Z 624.382,A -85,B 0,C 180,E1 -13047.766,E2 -13047.766} C_VEL
LIN {X 0,Y 360.539,Z 625.267,A -85,B 0,C 180,E1 -13048.883,E2 -13048.883} C_VEL
LIN {X 0,Y 360.528,Z 625.737,A -85,B 0,C 180,E1 -13050,E2 -13050} C_VEL
LIN {X 0,Y 360.53,Z 625.743,A -85,B 0,C 180,E1 -13051.117,E2 -13051.117} C_VEL
LIN {X 0,Y 360.47,Z 625.321,A -85,B 0,C 180,E1 -13052.235,E2 -13052.235} C_VEL
LIN {X 0,Y 360.379,Z 624.492,A -85,B 0,C 180,E1 -13053.354,E2 -13053.354} C_VEL
LIN {X 0,Y 360.414,Z 623.251,A -85,B 0,C 180,E1 -13054.474,E2 -13054.474} C_VEL
LIN {X 0,Y 360.388,Z 620.858,A -85,B 0,C 180,E1 -13055.978,E2 -13055.978} C_VEL
LIN {X 0,Y 360.658,Z 616.813,A -85,B 0,C 180,E1 -13057.84,E2 -13057.84} C_VEL
LIN {X 0,Y 361.013,Z 612,A -85,B 0,C 180,E1 -13059.525,E2 -13059.525} C_VEL
LIN {X 0,Y 361.732,Z 604.84,A -85,B 0,C 180,E1 -13061.487,E2 -13061.487} C_VEL
LIN {X 0,Y 362.702,Z 597.212,A -85,B 0,C 180,E1 -13063.16,E2 -13063.16} C_VEL
LIN {X 0,Y 363.777,Z 588.057,A -85,B 0,C 180,E1 -13064.814,E2 -13064.814} C_VEL
LIN {X 0,Y 365.317,Z 577.52,A -85,B 0,C 180,E1 -13066.341,E2 -13066.341} C_VEL
LIN {X 0,Y 366.928,Z 566.055,A -85,B 0,C 180,E1 -13067.702,E2 -13067.702} C_VEL
LIN {X 0,Y 367.783,Z 557.856,A -85,B 0,C 180,E1 -13068.523,E2 -13068.523} C_VEL
LIN {X 0,Y 367.583,Z 544.69,A -85,B 0,C 180,E1 -13069.744,E2 -13069.744} C_VEL
LIN {X 0,Y 365.977,Z 532.807,A -85,B 0,C 180,E1 -13070.757,E2 -13070.757} C_VEL
LIN {X 0,Y 363.314,Z 521.241,A -85,B 0,C 180,E1 -13071.715,E2 -13071.715} C_VEL
LIN {X 0,Y 361.53,Z 514.575,A -85,B 0,C 180,E1 -13072.258,E2 -13072.258} C_VEL
LIN {X 0,Y 362.194,Z 507.604,A -85,B 0,C 180,E1 -13075.887,E2 -13075.887} C_VEL
LIN {X 0,Y 362.987,Z 501.381,A -85,B 0,C 180,E1 -13079.393,E2 -13079.393} C_VEL
LIN {X 0,Y 363.881,Z 496.022,A -85,B 0,C 180,E1 -13082.738,E2 -13082.738} C_VEL
LIN {X 0,Y 364.56,Z 492.338,A -85,B 0,C 180,E1 -13085.334,E2 -13085.334} C_VEL
LIN {X 0,Y 364.845,Z 489.292,A -85,B 0,C 180,E1 -13087.835,E2 -13087.835} C_VEL
LIN {X 0,Y 364.662,Z 487.532,A -85,B 0,C 180,E1 -13089.565,E2 -13089.565} C_VEL
LIN {X 0,Y 364.242,Z 484.838,A -85,B 0,C 180,E1 -13092.844,E2 -13092.844} C_VEL
LIN {X 0,Y 363.951,Z 483.021,A -85,B 0,C 180,E1 -13095.959,E2 -13095.959} C_VEL
LIN {X 0,Y 363.679,Z 481.94,A -85,B 0,C 180,E1 -13098.926,E2 -13098.926} C_VEL
LIN {X 0,Y 363.457,Z 481.393,A -85,B 0,C 180,E1 -13102.448,E2 -13102.448} C_VEL
LIN {X 0,Y 363.296,Z 481.431,A -85,B 0,C 180,E1 -13104.525,E2 -13104.525} C_VEL
LIN {X 0,Y 362.987,Z 481.817,A -85,B 0,C 180,E1 -13107.172,E2 -13107.172} C_VEL
LIN {X 0,Y 362.66,Z 482.509,A -85,B 0,C 180,E1 -13109.745,E2 -13109.745} C_VEL
LIN {X 0,Y 362.172,Z 483.969,A -85,B 0,C 180,E1 -13113.492,E2 -13113.492} C_VEL
LIN {X 0,Y 361.826,Z 485.789,A -85,B 0,C 180,E1 -13117.141,E2 -13117.141} C_VEL
LIN {X 0,Y 361.788,Z 486.293,A -85,B 0,C 180,E1 -13117.957,E2 -13117.957} C_VEL
LIN {X 0,Y 362.879,Z 489.187,A -85,B 0,C 180,E1 -13118.245,E2 -13118.245} C_VEL
LIN {X 0,Y 367.039,Z 498.796,A -85,B 0,C 180,E1 -13119.298,E2 -13119.298} C_VEL
LIN {X 0,Y 370.395,Z 510.16,A -85,B 0,C 180,E1 -13120.511,E2 -13120.511} C_VEL
LIN {X 0,Y 370.851,Z 511.933,A -85,B 0,C 180,E1 -13120.704,E2 -13120.704} C_VEL
LIN {X 0,Y 369.645,Z 523.855,A -85,B 0,C 180,E1 -13121.774,E2 -13121.774} C_VEL
LIN {X 0,Y 368.141,Z 535.378,A -85,B 0,C 180,E1 -13123.051,E2 -13123.051} C_VEL
LIN {X 0,Y 366.678,Z 545.501,A -85,B 0,C 180,E1 -13124.435,E2 -13124.435} C_VEL
LIN {X 0,Y 365.343,Z 553.765,A -85,B 0,C 180,E1 -13125.803,E2 -13125.803} C_VEL
LIN {X 0,Y 364.124,Z 561.913,A -85,B 0,C 180,E1 -13127.459,E2 -13127.459} C_VEL
LIN {X 0,Y 363.027,Z 569.43,A -85,B 0,C 180,E1 -13129.402,E2 -13129.402} C_VEL
LIN {X 0,Y 362.217,Z 574.551,A -85,B 0,C 180,E1 -13131.071,E2 -13131.071} C_VEL
LIN {X 0,Y 361.516,Z 578.788,A -85,B 0,C 180,E1 -13132.863,E2 -13132.863} C_VEL
LIN {X 0,Y 361.14,Z 581.463,A -85,B 0,C 180,E1 -13134.416,E2 -13134.416} C_VEL
LIN {X 0,Y 361.073,Z 582.881,A -85,B 0,C 180,E1 -13135.535,E2 -13135.535} C_VEL
LIN {X 0,Y 360.864,Z 583.877,A -85,B 0,C 180,E1 -13136.651,E2 -13136.651} C_VEL
LIN {X 0,Y 360.707,Z 584.46,A -85,B 0,C 180,E1 -13137.767,E2 -13137.767} C_VEL
LIN {X 0,Y 360.59,Z 584.65,A -85,B 0,C 180,E1 -13138.883,E2 -13138.883} C_VEL
LIN {X 0,Y 360.53,Z 584.441,A -85,B 0,C 180,E1 -13140,E2 -13140} C_VEL
LIN {X 0,Y 360.549,Z 583.78,A -85,B 0,C 180,E1 -13141.117,E2 -13141.117} C_VEL
LIN {X 0,Y 360.612,Z 582.71,A -85,B 0,C 180,E1 -13142.234,E2 -13142.234} C_VEL
LIN {X 0,Y 360.607,Z 581.24,A -85,B 0,C 180,E1 -13143.352,E2 -13143.352} C_VEL
LIN {X 0,Y 360.751,Z 578.186,A -85,B 0,C 180,E1 -13145.03,E2 -13145.03} C_VEL
LIN {X 0,Y 361.04,Z 573.56,A -85,B 0,C 180,E1 -13146.894,E2 -13146.894} C_VEL
LIN {X 0,Y 361.37,Z 567.776,A -85,B 0,C 180,E1 -13148.669,E2 -13148.669} C_VEL
LIN {X 0,Y 361.898,Z 560.915,A -85,B 0,C 180,E1 -13150.349,E2 -13150.349} C_VEL
LIN {X 0,Y 362.575,Z 552.453,A -85,B 0,C 180,E1 -13152.027,E2 -13152.027} C_VEL
LIN {X 0,Y 363.328,Z 543.811,A -85,B 0,C 180,E1 -13153.422,E2 -13153.422} C_VEL
LIN {X 0,Y 364.317,Z 532.254,A -85,B 0,C 180,E1 -13154.938,E2 -13154.938} C_VEL
LIN {X 0,Y 365.05,Z 521.57,A -85,B 0,C 180,E1 -13156.067,E2 -13156.067} C_VEL
LIN {X 0,Y 365.808,Z 510.128,A -85,B 0,C 180,E1 -13157.035,E2 -13157.035} C_VEL
LIN {X 0,Y 366.021,Z 505.331,A -85,B 0,C 180,E1 -13157.383,E2 -13157.383} C_VEL
LIN {X 0,Y 363.252,Z 492.196,A -85,B 0,C 180,E1 -13158.287,E2 -13158.287} C_VEL
LIN {X 0,Y 360.724,Z 480.007,A -85,B 0,C 180,E1 -13158.936,E2 -13158.936} C_VEL
LIN {X 0,Y 360.762,Z 476.05,A -85,B 0,C 180,E1 -13162.931,E2 -13162.931} C_VEL
LIN {X 0,Y 360.904,Z 472.501,A -85,B 0,C 180,E1 -13166.609,E2 -13166.609} C_VEL
LIN {X 0,Y 360.942,Z 471.53,A -85,B 0,C 180,E1 -13167.86,E2 -13167.86} C_VEL
LIN {X 0,Y 361.298,Z 471.479,A -85,B 0,C 180,E1 -13171.141,E2 -13171.141} C_VEL
LIN {X 0,Y 361.634,Z 471.441,A -85,B 0,C 180,E1 -13174.305,E2 -13174.305} C_VEL
LIN {X 0,Y 361.838,Z 471.411,A -85,B 0,C 180,E1 -13177.217,E2 -13177.217} C_VEL
LIN {X 0,Y 361.858,Z 471.41,A -85,B 0,C 180,E1 -13179.862,E2 -13179.862} C_VEL
LIN {X 0,Y 361.84,Z 471.411,A -85,B 0,C 180,E1 -13182.829,E2 -13182.829} C_VEL
LIN {X 0,Y 361.823,Z 471.416,A -85,B 0,C 180,E1 -13185.947,E2 -13185.947} C_VEL
LIN {X 0,Y 361.84,Z 471.41,A -85,B 0,C 180,E1 -13189.245,E2 -13189.245} C_VEL
LIN {X 0,Y 361.875,Z 471.406,A -85,B 0,C 180,E1 -13192.776,E2 -13192.776} C_VEL
LIN {X 0,Y 361.859,Z 471.409,A -85,B 0,C 180,E1 -13195.72,E2 -13195.72} C_VEL
LIN {X 0,Y 361.879,Z 471.407,A -85,B 0,C 180,E1 -13199.672,E2 -13199.672} C_VEL
LIN {X 0,Y 361.959,Z 471.396,A -85,B 0,C 180,E1 -13203.475,E2 -13203.475} C_VEL
LIN {X 0,Y 361.895,Z 471.403,A -85,B 0,C 180,E1 -13207.145,E2 -13207.145} C_VEL
LIN {X 0,Y 361.926,Z 471.401,A -85,B 0,C 180,E1 -13210.724,E2 -13210.724} C_VEL
LIN {X 0,Y 361.951,Z 471.401,A -85,B 0,C 180,E1 -13214.226,E2 -13214.226} C_VEL
LIN {X 0,Y 362.004,Z 471.391,A -85,B 0,C 180,E1 -13216.528,E2 -13216.528} C_VEL
LIN {X 0,Y 362.036,Z 471.39,A -85,B 0,C 180,E1 -13219.938,E2 -13219.938} C_VEL
LIN {X 0,Y 362.157,Z 471.375,A -85,B 0,C 180,E1 -13222.193,E2 -13222.193} C_VEL
LIN {X 0,Y 362.123,Z 471.378,A -85,B 0,C 180,E1 -13224.431,E2 -13224.431} C_VEL
LIN {X 0,Y 362.286,Z 471.358,A -85,B 0,C 180,E1 -13227.776,E2 -13227.776} C_VEL
LIN {X 0,Y 362.432,Z 471.342,A -85,B 0,C 180,E1 -13230,E2 -13230} C_VEL
LIN {X 0,Y 362.286,Z 471.358,A -85,B 0,C 180,E1 -13232.224,E2 -13232.224} C_VEL
LIN {X 0,Y 362.141,Z 471.374,A -85,B 0,C 180,E1 -13236.687,E2 -13236.687} C_VEL
LIN {X 0,Y 362.033,Z 471.391,A -85,B 0,C 180,E1 -13240.062,E2 -13240.062} C_VEL
LIN {X 0,Y 362.003,Z 471.395,A -85,B 0,C 180,E1 -13243.899,E2 -13243.899} C_VEL
LIN {X 0,Y 361.972,Z 471.398,A -85,B 0,C 180,E1 -13247.939,E2 -13247.939} C_VEL
LIN {X 0,Y 361.885,Z 471.409,A -85,B 0,C 180,E1 -13251.653,E2 -13251.653} C_VEL
LIN {X 0,Y 361.931,Z 471.4,A -85,B 0,C 180,E1 -13255.29,E2 -13255.29} C_VEL
LIN {X 0,Y 361.913,Z 471.406,A -85,B 0,C 180,E1 -13257.779,E2 -13257.779} C_VEL
LIN {X 0,Y 361.842,Z 471.414,A -85,B 0,C 180,E1 -13261.629,E2 -13261.629} C_VEL
LIN {X 0,Y 361.879,Z 471.407,A -85,B 0,C 180,E1 -13265.345,E2 -13265.345} C_VEL
LIN {X 0,Y 361.875,Z 471.405,A -85,B 0,C 180,E1 -13269.027,E2 -13269.027} C_VEL
LIN {X 0,Y 361.84,Z 471.41,A -85,B 0,C 180,E1 -13272.828,E2 -13272.828} C_VEL
LIN {X 0,Y 361.821,Z 471.417,A -85,B 0,C 180,E1 -13275.602,E2 -13275.602} C_VEL
LIN {X 0,Y 361.19,Z 471.5,A -85,B 0,C 180,E1 -13276.532,E2 -13276.532} C_VEL
LIN {X 0,Y 358.311,Z 471.854,A -85,B 0,C 180,E1 -13278.044,E2 -13278.044} C_VEL
LIN {X 0,Y 355.877,Z 472.155,A -85,B 0,C 180,E1 -13279.267,E2 -13279.267} C_VEL
LIN {X 0,Y 354.878,Z 472.278,A -85,B 0,C 180,E1 -13280.214,E2 -13280.214} C_VEL
LIN {X 0,Y 354.823,Z 472.283,A -85,B 0,C 180,E1 -13280.534,E2 -13280.534} C_VEL
LIN {X 0,Y 354.766,Z 472.295,A -85,B 0,C 180,E1 -13283.536,E2 -13283.536} C_VEL
LIN {X 0,Y 354.628,Z 472.309,A -85,B 0,C 180,E1 -13286.342,E2 -13286.342} C_VEL
LIN {X 0,Y 354.314,Z 472.349,A -85,B 0,C 180,E1 -13288.954,E2 -13288.954} C_VEL
LIN {X 0,Y 353.995,Z 472.393,A -85,B 0,C 180,E1 -13291.544,E2 -13291.544} C_VEL
LIN {X 0,Y 353.693,Z 472.431,A -85,B 0,C 180,E1 -13294.078,E2 -13294.078} C_VEL
LIN {X 0,Y 353.574,Z 476.376,A -85,B 0,C 180,E1 -13297.811,E2 -13297.811} C_VEL
LIN {X 0,Y 353.594,Z 479.837,A -85,B 0,C 180,E1 -13300.969,E2 -13300.969} C_VEL
LIN {X 0,Y 356.38,Z 493.619,A -85,B 0,C 180,E1 -13301.705,E2 -13301.705} C_VEL
LIN {X 0,Y 358.874,Z 505.895,A -85,B 0,C 180,E1 -13302.573,E2 -13302.573} C_VEL
LIN {X 0,Y 358.33,Z 517.214,A -85,B 0,C 180,E1 -13303.477,E2 -13303.477} C_VEL
LIN {X 0,Y 357.568,Z 528.995,A -85,B 0,C 180,E1 -13304.653,E2 -13304.653} C_VEL
LIN {X 0,Y 356.569,Z 540.038,A -85,B 0,C 180,E1 -13306.028,E2 -13306.028} C_VEL
LIN {X 0,Y 355.746,Z 549.385,A -85,B 0,C 180,E1 -13307.448,E2 -13307.448} C_VEL
LIN {X 0,Y 355.017,Z 558.486,A -85,B 0,C 180,E1 -13309.16,E2 -13309.16} C_VEL
LIN {X 0,Y 354.394,Z 565.869,A -85,B 0,C 180,E1 -13310.871,E2 -13310.871} C_VEL
LIN {X 0,Y 353.995,Z 571.808,A -85,B 0,C 180,E1 -13312.585,E2 -13312.585} C_VEL
LIN {X 0,Y 353.74,Z 576.479,A -85,B 0,C 180,E1 -13314.299,E2 -13314.299} C_VEL
LIN {X 0,Y 353.534,Z 580.036,A -85,B 0,C 180,E1 -13316.01,E2 -13316.01} C_VEL
LIN {X 0,Y 353.511,Z 582.572,A -85,B 0,C 180,E1 -13317.721,E2 -13317.721} C_VEL
LIN {X 0,Y 353.46,Z 583.71,A -85,B 0,C 180,E1 -13318.86,E2 -13318.86} C_VEL
LIN {X 0,Y 353.456,Z 584.448,A -85,B 0,C 180,E1 -13320,E2 -13320} C_VEL
LIN {X 0,Y 353.507,Z 584.782,A -85,B 0,C 180,E1 -13321.139,E2 -13321.139} C_VEL
LIN {X 0,Y 353.637,Z 584.662,A -85,B 0,C 180,E1 -13322.278,E2 -13322.278} C_VEL
LIN {X 0,Y 353.817,Z 584.147,A -85,B 0,C 180,E1 -13323.416,E2 -13323.416} C_VEL
LIN {X 0,Y 354.005,Z 583.246,A -85,B 0,C 180,E1 -13324.554,E2 -13324.554} C_VEL
LIN {X 0,Y 354.014,Z 581.92,A -85,B 0,C 180,E1 -13325.696,E2 -13325.696} C_VEL
LIN {X 0,Y 354.709,Z 578.221,A -85,B 0,C 180,E1 -13327.831,E2 -13327.831} C_VEL
LIN {X 0,Y 355.436,Z 573.752,A -85,B 0,C 180,E1 -13329.675,E2 -13329.675} C_VEL
LIN {X 0,Y 356.52,Z 567.37,A -85,B 0,C 180,E1 -13331.657,E2 -13331.657} C_VEL
LIN {X 0,Y 357.581,Z 560.487,A -85,B 0,C 180,E1 -13333.352,E2 -13333.352} C_VEL
LIN {X 0,Y 358.944,Z 551.981,A -85,B 0,C 180,E1 -13335.036,E2 -13335.036} C_VEL
LIN {X 0,Y 360.737,Z 541.476,A -85,B 0,C 180,E1 -13336.7,E2 -13336.7} C_VEL
LIN {X 0,Y 362.317,Z 530.401,A -85,B 0,C 180,E1 -13338.107,E2 -13338.107} C_VEL
LIN {X 0,Y 363.88,Z 518.913,A -85,B 0,C 180,E1 -13339.274,E2 -13339.274} C_VEL
LIN {X 0,Y 364.343,Z 513.27,A -85,B 0,C 180,E1 -13339.779,E2 -13339.779} C_VEL
LIN {X 0,Y 361.98,Z 503.396,A -85,B 0,C 180,E1 -13340.874,E2 -13340.874} C_VEL
LIN {X 0,Y 357.96,Z 492.665,A -85,B 0,C 180,E1 -13342.086,E2 -13342.086} C_VEL
LIN {X 0,Y 355.57,Z 487.658,A -85,B 0,C 180,E1 -13342.68,E2 -13342.68} C_VEL
LIN {X 0,Y 354.743,Z 485.178,A -85,B 0,C 180,E1 -13342.947,E2 -13342.947} C_VEL
LIN {X 0,Y 354.963,Z 481.435,A -85,B 0,C 180,E1 -13347.004,E2 -13347.004} C_VEL
LIN {X 0,Y 355.161,Z 477.923,A -85,B 0,C 180,E1 -13350.963,E2 -13350.963} C_VEL
LIN {X 0,Y 355.23,Z 475.596,A -85,B 0,C 180,E1 -13353.804,E2 -13353.804} C_VEL
LIN {X 0,Y 355.077,Z 473.632,A -85,B 0,C 180,E1 -13356.426,E2 -13356.426} C_VEL
LIN {X 0,Y 354.836,Z 472.286,A -85,B 0,C 180,E1 -13358.601,E2 -13358.601} C_VEL
LIN {X 0,Y 354.796,Z 472.292,A -85,B 0,C 180,E1 -13362.337,E2 -13362.337} C_VEL
LIN {X 0,Y 354.864,Z 472.437,A -85,B 0,C 180,E1 -13365.477,E2 -13365.477} C_VEL
LIN {X 0,Y 356.026,Z 478.784,A -85,B 0,C 180,E1 -13369.351,E2 -13369.351} C_VEL
LIN {X 0,Y 357.063,Z 485.292,A -85,B 0,C 180,E1 -13373.107,E2 -13373.107} C_VEL
LIN {X 0,Y 356.925,Z 489.111,A -85,B 0,C 180,E1 -13375.178,E2 -13375.178} C_VEL
LIN {X 0,Y 356.106,Z 495.601,A -85,B 0,C 180,E1 -13378.579,E2 -13378.579} C_VEL
LIN {X 0,Y 355.358,Z 502.871,A -85,B 0,C 180,E1 -13382.305,E2 -13382.305} C_VEL
LIN {X 0,Y 354.675,Z 509.672,A -85,B 0,C 180,E1 -13385.714,E2 -13385.714} C_VEL
LIN {X 0,Y 354.424,Z 512.821,A -85,B 0,C 180,E1 -13387.279,E2 -13387.279} C_VEL
LIN {X 0,Y 355.207,Z 516.593,A -85,B 0,C 180,E1 -13387.57,E2 -13387.57} C_VEL
LIN {X 0,Y 357.199,Z 524.492,A -85,B 0,C 180,E1 -13388.233,E2 -13388.233} C_VEL
LIN {X 0,Y 359.497,Z 536.709,A -85,B 0,C 180,E1 -13389.292,E2 -13389.292} C_VEL
LIN {X 0,Y 360.436,Z 546.452,A -85,B 0,C 180,E1 -13390.176,E2 -13390.176} C_VEL
LIN {X 0,Y 360.648,Z 560.081,A -85,B 0,C 180,E1 -13391.538,E2 -13391.538} C_VEL
LIN {X 0,Y 359.066,Z 571.236,A -85,B 0,C 180,E1 -13392.78,E2 -13392.78} C_VEL
LIN {X 0,Y 357.509,Z 582.368,A -85,B 0,C 180,E1 -13394.296,E2 -13394.296} C_VEL
LIN {X 0,Y 356.324,Z 590.947,A -85,B 0,C 180,E1 -13395.727,E2 -13395.727} C_VEL
LIN {X 0,Y 355.214,Z 599.312,A -85,B 0,C 180,E1 -13397.43,E2 -13397.43} C_VEL
LIN {X 0,Y 354.351,Z 606.227,A -85,B 0,C 180,E1 -13399.139,E2 -13399.139} C_VEL
LIN {X 0,Y 353.817,Z 611.816,A -85,B 0,C 180,E1 -13400.857,E2 -13400.857} C_VEL
LIN {X 0,Y 353.513,Z 616.221,A -85,B 0,C 180,E1 -13402.575,E2 -13402.575} C_VEL
LIN {X 0,Y 353.404,Z 619.564,A -85,B 0,C 180,E1 -13404.293,E2 -13404.293} C_VEL
LIN {X 0,Y 353.385,Z 621.245,A -85,B 0,C 180,E1 -13405.437,E2 -13405.437} C_VEL
LIN {X 0,Y 353.477,Z 623.816,A -85,B 0,C 180,E1 -13407.721,E2 -13407.721} C_VEL
LIN {X 0,Y 353.476,Z 624.737,A -85,B 0,C 180,E1 -13408.861,E2 -13408.861} C_VEL
LIN {X 0,Y 353.463,Z 625.243,A -85,B 0,C 180,E1 -13410,E2 -13410} C_VEL
LIN {X 0,Y 353.464,Z 625.318,A -85,B 0,C 180,E1 -13411.139,E2 -13411.139} C_VEL
LIN {X 0,Y 353.371,Z 624.931,A -85,B 0,C 180,E1 -13412.28,E2 -13412.28} C_VEL
LIN {X 0,Y 353.321,Z 622.937,A -85,B 0,C 180,E1 -13414.564,E2 -13414.564} C_VEL
LIN {X 0,Y 353.314,Z 620.847,A -85,B 0,C 180,E1 -13415.966,E2 -13415.966} C_VEL
LIN {X 0,Y 353.604,Z 616.652,A -85,B 0,C 180,E1 -13417.997,E2 -13417.997} C_VEL
LIN {X 0,Y 353.981,Z 611.939,A -85,B 0,C 180,E1 -13419.716,E2 -13419.716} C_VEL
LIN {X 0,Y 354.771,Z 604.944,A -85,B 0,C 180,E1 -13421.716,E2 -13421.716} C_VEL
LIN {X 0,Y 355.788,Z 597.462,A -85,B 0,C 180,E1 -13423.421,E2 -13423.421} C_VEL
LIN {X 0,Y 356.861,Z 588.947,A -85,B 0,C 180,E1 -13425.027,E2 -13425.027} C_VEL
LIN {X 0,Y 358.551,Z 578.255,A -85,B 0,C 180,E1 -13426.659,E2 -13426.659} C_VEL
LIN {X 0,Y 360.236,Z 567.146,A -85,B 0,C 180,E1 -13428.042,E2 -13428.042} C_VEL
LIN {X 0,Y 361.217,Z 559.298,A -85,B 0,C 180,E1 -13428.873,E2 -13428.873} C_VEL
LIN {X 0,Y 361.195,Z 546.77,A -85,B 0,C 180,E1 -13430.098,E2 -13430.098} C_VEL
LIN {X 0,Y 359.755,Z 534.696,A -85,B 0,C 180,E1 -13431.215,E2 -13431.215} C_VEL
LIN {X 0,Y 357.159,Z 523.02,A -85,B 0,C 180,E1 -13432.246,E2 -13432.246} C_VEL
LIN {X 0,Y 355.356,Z 517.04,A -85,B 0,C 180,E1 -13432.792,E2 -13432.792} C_VEL
LIN {X 0,Y 354.615,Z 513.908,A -85,B 0,C 180,E1 -13433.054,E2 -13433.054} C_VEL
LIN {X 0,Y 355.281,Z 507.666,A -85,B 0,C 180,E1 -13436.429,E2 -13436.429} C_VEL
LIN {X 0,Y 356.056,Z 502.051,A -85,B 0,C 180,E1 -13439.716,E2 -13439.716} C_VEL
LIN {X 0,Y 356.726,Z 498.244,A -85,B 0,C 180,E1 -13442.137,E2 -13442.137} C_VEL
LIN {X 0,Y 357.444,Z 494.507,A -85,B 0,C 180,E1 -13444.764,E2 -13444.764} C_VEL
LIN {X 0,Y 357.795,Z 492.467,A -85,B 0,C 180,E1 -13446.356,E2 -13446.356} C_VEL
LIN {X 0,Y 357.779,Z 489.641,A -85,B 0,C 180,E1 -13448.946,E2 -13448.946} C_VEL
LIN {X 0,Y 357.413,Z 487.045,A -85,B 0,C 180,E1 -13451.956,E2 -13451.956} C_VEL
LIN {X 0,Y 357.085,Z 485.014,A -85,B 0,C 180,E1 -13455.116,E2 -13455.116} C_VEL
LIN {X 0,Y 356.777,Z 483.627,A -85,B 0,C 180,E1 -13458.465,E2 -13458.465} C_VEL
LIN {X 0,Y 356.56,Z 482.938,A -85,B 0,C 180,E1 -13462.039,E2 -13462.039} C_VEL
LIN {X 0,Y 356.268,Z 482.955,A -85,B 0,C 180,E1 -13465.105,E2 -13465.105} C_VEL
LIN {X 0,Y 355.924,Z 483.444,A -85,B 0,C 180,E1 -13468.111,E2 -13468.111} C_VEL
LIN {X 0,Y 355.415,Z 484.535,A -85,B 0,C 180,E1 -13471.668,E2 -13471.668} C_VEL
LIN {X 0,Y 354.985,Z 486.226,A -85,B 0,C 180,E1 -13475.604,E2 -13475.604} C_VEL
LIN {X 0,Y 354.855,Z 487.017,A -85,B 0,C 180,E1 -13477.145,E2 -13477.145} C_VEL
LIN {X 0,Y 355.852,Z 489.82,A -85,B 0,C 180,E1 -13477.438,E2 -13477.438} C_VEL
LIN {X 0,Y 357.989,Z 494.026,A -85,B 0,C 180,E1 -13477.965,E2 -13477.965} C_VEL
LIN {X 0,Y 361.931,Z 504.222,A -85,B 0,C 180,E1 -13479.157,E2 -13479.157} C_VEL
LIN {X 0,Y 364.472,Z 513.794,A -85,B 0,C 180,E1 -13480.259,E2 -13480.259} C_VEL
LIN {X 0,Y 364.371,Z 516.971,A -85,B 0,C 180,E1 -13480.556,E2 -13480.556} C_VEL
LIN {X 0,Y 362.82,Z 528.599,A -85,B 0,C 180,E1 -13481.69,E2 -13481.69} C_VEL
LIN {X 0,Y 361.248,Z 539.614,A -85,B 0,C 180,E1 -13483.033,E2 -13483.033} C_VEL
LIN {X 0,Y 359.733,Z 548.87,A -85,B 0,C 180,E1 -13484.417,E2 -13484.417} C_VEL
LIN {X 0,Y 358.425,Z 556.592,A -85,B 0,C 180,E1 -13485.812,E2 -13485.812} C_VEL
LIN {X 0,Y 357.08,Z 564.286,A -85,B 0,C 180,E1 -13487.497,E2 -13487.497} C_VEL
LIN {X 0,Y 356.142,Z 570.487,A -85,B 0,C 180,E1 -13489.195,E2 -13489.195} C_VEL
LIN {X 0,Y 355.272,Z 575.452,A -85,B 0,C 180,E1 -13490.895,E2 -13490.895} C_VEL
LIN {X 0,Y 354.488,Z 579.712,A -85,B 0,C 180,E1 -13492.792,E2 -13492.792} C_VEL
LIN {X 0,Y 354.1,Z 582.167,A -85,B 0,C 180,E1 -13494.305,E2 -13494.305} C_VEL
LIN {X 0,Y 354.036,Z 583.522,A -85,B 0,C 180,E1 -13495.446,E2 -13495.446} C_VEL
LIN {X 0,Y 353.82,Z 584.446,A -85,B 0,C 180,E1 -13496.584,E2 -13496.584} C_VEL
LIN {X 0,Y 353.65,Z 584.978,A -85,B 0,C 180,E1 -13497.722,E2 -13497.722} C_VEL
LIN {X 0,Y 353.526,Z 585.118,A -85,B 0,C 180,E1 -13498.861,E2 -13498.861} C_VEL
LIN {X 0,Y 353.465,Z 584.834,A -85,B 0,C 180,E1 -13500,E2 -13500} C_VEL
LIN {X 0,Y 353.486,Z 584.117,A -85,B 0,C 180,E1 -13501.14,E2 -13501.14} C_VEL
LIN {X 0,Y 353.518,Z 583.003,A -85,B 0,C 180,E1 -13502.279,E2 -13502.279} C_VEL
LIN {X 0,Y 353.539,Z 580.526,A -85,B 0,C 180,E1 -13503.99,E2 -13503.99} C_VEL
LIN {X 0,Y 353.756,Z 577.033,A -85,B 0,C 180,E1 -13505.701,E2 -13505.701} C_VEL
LIN {X 0,Y 354.049,Z 572.439,A -85,B 0,C 180,E1 -13507.413,E2 -13507.413} C_VEL
LIN {X 0,Y 354.437,Z 566.619,A -85,B 0,C 180,E1 -13509.128,E2 -13509.128} C_VEL
LIN {X 0,Y 355.009,Z 559.372,A -85,B 0,C 180,E1 -13510.84,E2 -13510.84} C_VEL
LIN {X 0,Y 355.73,Z 550.381,A -85,B 0,C 180,E1 -13512.552,E2 -13512.552} C_VEL
LIN {X 0,Y 356.655,Z 540.246,A -85,B 0,C 180,E1 -13514.114,E2 -13514.114} C_VEL
LIN {X 0,Y 357.474,Z 529.944,A -85,B 0,C 180,E1 -13515.402,E2 -13515.402} C_VEL
LIN {X 0,Y 358.341,Z 517.407,A -85,B 0,C 180,E1 -13516.669,E2 -13516.669} C_VEL
LIN {X 0,Y 359.063,Z 507.592,A -85,B 0,C 180,E1 -13517.458,E2 -13517.458} C_VEL
LIN {X 0,Y 357.067,Z 496.682,A -85,B 0,C 180,E1 -13518.254,E2 -13518.254} C_VEL
LIN {X 0,Y 354.036,Z 482.545,A -85,B 0,C 180,E1 -13519.063,E2 -13519.063} C_VEL
LIN {X 0,Y 353.631,Z 480.363,A -85,B 0,C 180,E1 -13519.199,E2 -13519.199} C_VEL
LIN {X 0,Y 353.638,Z 477.42,A -85,B 0,C 180,E1 -13522.185,E2 -13522.185} C_VEL
LIN {X 0,Y 353.809,Z 473.84,A -85,B 0,C 180,E1 -13525.913,E2 -13525.913} C_VEL
LIN {X 0,Y 353.84,Z 472.639,A -85,B 0,C 180,E1 -13527.183,E2 -13527.183} C_VEL
LIN {X 0,Y 354.095,Z 472.38,A -85,B 0,C 180,E1 -13529.749,E2 -13529.749} C_VEL
LIN {X 0,Y 354.393,Z 472.343,A -85,B 0,C 180,E1 -13532.374,E2 -13532.374} C_VEL
LIN {X 0,Y 354.715,Z 472.299,A -85,B 0,C 180,E1 -13535.675,E2 -13535.675} C_VEL
LIN {X 0,Y 354.796,Z 472.29,A -85,B 0,C 180,E1 -13537.885,E2 -13537.885} C_VEL
LIN {X 0,Y 354.792,Z 472.287,A -85,B 0,C 180,E1 -13541.172,E2 -13541.172} C_VEL
LIN {X 0,Y 354.769,Z 472.295,A -85,B 0,C 180,E1 -13544.507,E2 -13544.507} C_VEL
LIN {X 0,Y 354.798,Z 472.289,A -85,B 0,C 180,E1 -13547.663,E2 -13547.663} C_VEL
LIN {X 0,Y 354.819,Z 472.287,A -85,B 0,C 180,E1 -13550.666,E2 -13550.666} C_VEL
LIN {X 0,Y 354.826,Z 472.288,A -85,B 0,C 180,E1 -13554.301,E2 -13554.301} C_VEL
LIN {X 0,Y 354.792,Z 472.29,A -85,B 0,C 180,E1 -13557.667,E2 -13557.667} C_VEL
LIN {X 0,Y 354.873,Z 472.28,A -85,B 0,C 180,E1 -13560.622,E2 -13560.622} C_VEL
LIN {X 0,Y 354.904,Z 472.279,A -85,B 0,C 180,E1 -13564.173,E2 -13564.173} C_VEL
LIN {X 0,Y 354.839,Z 472.286,A -85,B 0,C 180,E1 -13567.894,E2 -13567.894} C_VEL
LIN {X 0,Y 354.928,Z 472.275,A -85,B 0,C 180,E1 -13571.891,E2 -13571.891} C_VEL
LIN {X 0,Y 354.948,Z 472.273,A -85,B 0,C 180,E1 -13575.981,E2 -13575.981} C_VEL
LIN {X 0,Y 354.983,Z 472.267,A -85,B 0,C 180,E1 -13579.736,E2 -13579.736} C_VEL
LIN {X 0,Y 355.12,Z 472.252,A -85,B 0,C 180,E1 -13582.037,E2 -13582.037} C_VEL
LIN {X 0,Y 355.097,Z 472.253,A -85,B 0,C 180,E1 -13584.321,E2 -13584.321} C_VEL
LIN {X 0,Y 355.249,Z 472.235,A -85,B 0,C 180,E1 -13587.732,E2 -13587.732} C_VEL
LIN {X 0,Y 355.401,Z 472.217,A -85,B 0,C 180,E1 -13590,E2 -13590} C_VEL
LIN {X 0,Y 355.249,Z 472.234,A -85,B 0,C 180,E1 -13592.268,E2 -13592.268} C_VEL
LIN {X 0,Y 355.105,Z 472.249,A -85,B 0,C 180,E1 -13596.82,E2 -13596.82} C_VEL
LIN {X 0,Y 354.981,Z 472.267,A -85,B 0,C 180,E1 -13600.264,E2 -13600.264} C_VEL
LIN {X 0,Y 354.948,Z 472.273,A -85,B 0,C 180,E1 -13604.019,E2 -13604.019} C_VEL
LIN {X 0,Y 354.928,Z 472.275,A -85,B 0,C 180,E1 -13608.109,E2 -13608.109} C_VEL
LIN {X 0,Y 354.831,Z 472.287,A -85,B 0,C 180,E1 -13612.106,E2 -13612.106} C_VEL
LIN {X 0,Y 354.903,Z 472.279,A -85,B 0,C 180,E1 -13615.827,E2 -13615.827} C_VEL
LIN {X 0,Y 354.822,Z 472.289,A -85,B 0,C 180,E1 -13619.682,E2 -13619.682} C_VEL
LIN {X 0,Y 354.81,Z 472.29,A -85,B 0,C 180,E1 -13623.702,E2 -13623.702} C_VEL
LIN {X 0,Y 354.806,Z 472.287,A -85,B 0,C 180,E1 -13626.459,E2 -13626.459} C_VEL
LIN {X 0,Y 354.828,Z 472.286,A -85,B 0,C 180,E1 -13629.423,E2 -13629.423} C_VEL
LIN {X 0,Y 354.792,Z 472.288,A -85,B 0,C 180,E1 -13632.867,E2 -13632.867} C_VEL
LIN {X 0,Y 354.772,Z 472.293,A -85,B 0,C 180,E1 -13636.104,E2 -13636.104} C_VEL
LIN {X 0,Y 354.792,Z 472.289,A -85,B 0,C 180,E1 -13639.179,E2 -13639.179} C_VEL
LIN {X 0,Y 354.823,Z 472.283,A -85,B 0,C 180,E1 -13640.534,E2 -13640.534} C_VEL
LIN {X 0,Y 354.216,Z 472.365,A -85,B 0,C 180,E1 -13641.482,E2 -13641.482} C_VEL
LIN {X 0,Y 351.334,Z 472.73,A -85,B 0,C 180,E1 -13643.021,E2 -13643.021} C_VEL
LIN {X 0,Y 348.828,Z 473.04,A -85,B 0,C 180,E1 -13644.266,E2 -13644.266} C_VEL
LIN {X 0,Y 347.721,Z 473.174,A -85,B 0,C 180,E1 -13645.231,E2 -13645.231} C_VEL
LIN {X 0,Y 347.617,Z 473.186,A -85,B 0,C 180,E1 -13645.559,E2 -13645.559} C_VEL
LIN {X 0,Y 347.378,Z 473.213,A -85,B 0,C 180,E1 -13648.263,E2 -13648.263} C_VEL
LIN {X 0,Y 347.046,Z 473.254,A -85,B 0,C 180,E1 -13650.92,E2 -13650.92} C_VEL
LIN {X 0,Y 346.722,Z 473.299,A -85,B 0,C 180,E1 -13653.516,E2 -13653.516} C_VEL
LIN {X 0,Y 346.554,Z 473.763,A -85,B 0,C 180,E1 -13654.794,E2 -13654.794} C_VEL
LIN {X 0,Y 346.55,Z 478.184,A -85,B 0,C 180,E1 -13658.888,E2 -13658.888} C_VEL
LIN {X 0,Y 346.524,Z 480.237,A -85,B 0,C 180,E1 -13660.718,E2 -13660.718} C_VEL
LIN {X 0,Y 349.323,Z 493.993,A -85,B 0,C 180,E1 -13661.474,E2 -13661.474} C_VEL
LIN {X 0,Y 351.966,Z 507.651,A -85,B 0,C 180,E1 -13662.473,E2 -13662.473} C_VEL
LIN {X 0,Y 351.245,Z 519.169,A -85,B 0,C 180,E1 -13663.433,E2 -13663.433} C_VEL
LIN {X 0,Y 350.355,Z 531.251,A -85,B 0,C 180,E1 -13664.71,E2 -13664.71} C_VEL
LIN {X 0,Y 349.496,Z 541.435,A -85,B 0,C 180,E1 -13666.036,E2 -13666.036} C_VEL
LIN {X 0,Y 348.616,Z 550.58,A -85,B 0,C 180,E1 -13667.483,E2 -13667.483} C_VEL
LIN {X 0,Y 347.905,Z 559.553,A -85,B 0,C 180,E1 -13669.23,E2 -13669.23} C_VEL
LIN {X 0,Y 347.279,Z 566.828,A -85,B 0,C 180,E1 -13670.976,E2 -13670.976} C_VEL
LIN {X 0,Y 346.832,Z 573.471,A -85,B 0,C 180,E1 -13673.016,E2 -13673.016} C_VEL
LIN {X 0,Y 346.608,Z 577.861,A -85,B 0,C 180,E1 -13674.764,E2 -13674.764} C_VEL
LIN {X 0,Y 346.424,Z 581.164,A -85,B 0,C 180,E1 -13676.51,E2 -13676.51} C_VEL
LIN {X 0,Y 346.417,Z 582.828,A -85,B 0,C 180,E1 -13677.674,E2 -13677.674} C_VEL
LIN {X 0,Y 346.382,Z 584.021,A -85,B 0,C 180,E1 -13678.837,E2 -13678.837} C_VEL
LIN {X 0,Y 346.393,Z 584.809,A -85,B 0,C 180,E1 -13680,E2 -13680} C_VEL
LIN {X 0,Y 346.447,Z 585.207,A -85,B 0,C 180,E1 -13681.162,E2 -13681.162} C_VEL
LIN {X 0,Y 346.583,Z 585.166,A -85,B 0,C 180,E1 -13682.324,E2 -13682.324} C_VEL
LIN {X 0,Y 346.774,Z 584.698,A -85,B 0,C 180,E1 -13683.486,E2 -13683.486} C_VEL
LIN {X 0,Y 346.946,Z 583.843,A -85,B 0,C 180,E1 -13684.647,E2 -13684.647} C_VEL
LIN {X 0,Y 346.978,Z 582.61,A -85,B 0,C 180,E1 -13685.812,E2 -13685.812} C_VEL
LIN {X 0,Y 347.731,Z 579.085,A -85,B 0,C 180,E1 -13687.968,E2 -13687.968} C_VEL
LIN {X 0,Y 348.504,Z 574.695,A -85,B 0,C 180,E1 -13689.87,E2 -13689.87} C_VEL
LIN {X 0,Y 349.678,Z 568.472,A -85,B 0,C 180,E1 -13691.888,E2 -13691.888} C_VEL
LIN {X 0,Y 350.789,Z 561.771,A -85,B 0,C 180,E1 -13693.616,E2 -13693.616} C_VEL
LIN {X 0,Y 352.25,Z 553.553,A -85,B 0,C 180,E1 -13695.329,E2 -13695.329} C_VEL
LIN {X 0,Y 353.792,Z 545.166,A -85,B 0,C 180,E1 -13696.74,E2 -13696.74} C_VEL
LIN {X 0,Y 355.781,Z 532.831,A -85,B 0,C 180,E1 -13698.425,E2 -13698.425} C_VEL
LIN {X 0,Y 357.506,Z 521.451,A -85,B 0,C 180,E1 -13699.65,E2 -13699.65} C_VEL
LIN {X 0,Y 358.115,Z 515.196,A -85,B 0,C 180,E1 -13700.247,E2 -13700.247} C_VEL
LIN {X 0,Y 355.598,Z 504.88,A -85,B 0,C 180,E1 -13701.467,E2 -13701.467} C_VEL
LIN {X 0,Y 351.761,Z 494.745,A -85,B 0,C 180,E1 -13702.708,E2 -13702.708} C_VEL
LIN {X 0,Y 349.002,Z 488.949,A -85,B 0,C 180,E1 -13703.456,E2 -13703.456} C_VEL
LIN {X 0,Y 347.831,Z 485.877,A -85,B 0,C 180,E1 -13703.835,E2 -13703.835} C_VEL
LIN {X 0,Y 348.032,Z 482.767,A -85,B 0,C 180,E1 -13707.312,E2 -13707.312} C_VEL
LIN {X 0,Y 348.22,Z 480.231,A -85,B 0,C 180,E1 -13710.302,E2 -13710.302} C_VEL
LIN {X 0,Y 348.368,Z 478.077,A -85,B 0,C 180,E1 -13713.004,E2 -13713.004} C_VEL
LIN {X 0,Y 348.275,Z 475.8,A -85,B 0,C 180,E1 -13716.179,E2 -13716.179} C_VEL
LIN {X 0,Y 348.006,Z 474.254,A -85,B 0,C 180,E1 -13718.759,E2 -13718.759} C_VEL
LIN {X 0,Y 347.765,Z 473.168,A -85,B 0,C 180,E1 -13721.056,E2 -13721.056} C_VEL
LIN {X 0,Y 347.831,Z 473.229,A -85,B 0,C 180,E1 -13725.211,E2 -13725.211} C_VEL
LIN {X 0,Y 348.94,Z 479.497,A -85,B 0,C 180,E1 -13729.113,E2 -13729.113} C_VEL
LIN {X 0,Y 349.857,Z 484.86,A -85,B 0,C 180,E1 -13732.299,E2 -13732.299} C_VEL
LIN {X 0,Y 349.977,Z 488.555,A -85,B 0,C 180,E1 -13734.383,E2 -13734.383} C_VEL
LIN {X 0,Y 349.225,Z 494.696,A -85,B 0,C 180,E1 -13737.697,E2 -13737.697} C_VEL
LIN {X 0,Y 348.392,Z 502.3,A -85,B 0,C 180,E1 -13741.702,E2 -13741.702} C_VEL
LIN {X 0,Y 347.643,Z 509.621,A -85,B 0,C 180,E1 -13745.468,E2 -13745.468} C_VEL
LIN {X 0,Y 347.493,Z 511.521,A -85,B 0,C 180,E1 -13746.378,E2 -13746.378} C_VEL
LIN {X 0,Y 348.211,Z 515.083,A -85,B 0,C 180,E1 -13746.664,E2 -13746.664} C_VEL
LIN {X 0,Y 349.17,Z 518.417,A -85,B 0,C 180,E1 -13746.971,E2 -13746.971} C_VEL
LIN {X 0,Y 351.788,Z 529.6,A -85,B 0,C 180,E1 -13747.99,E2 -13747.99} C_VEL
LIN {X 0,Y 353.728,Z 542.452,A -85,B 0,C 180,E1 -13749.212,E2 -13749.212} C_VEL
LIN {X 0,Y 354.114,Z 554.736,A -85,B 0,C 180,E1 -13750.433,E2 -13750.433} C_VEL
LIN {X 0,Y 353.845,Z 562.766,A -85,B 0,C 180,E1 -13751.321,E2 -13751.321} C_VEL
LIN {X 0,Y 352.205,Z 573.395,A -85,B 0,C 180,E1 -13752.583,E2 -13752.583} C_VEL
LIN {X 0,Y 350.708,Z 583.166,A -85,B 0,C 180,E1 -13754.008,E2 -13754.008} C_VEL
LIN {X 0,Y 349.246,Z 592.849,A -85,B 0,C 180,E1 -13755.729,E2 -13755.729} C_VEL
LIN {X 0,Y 348.084,Z 600.834,A -85,B 0,C 180,E1 -13757.464,E2 -13757.464} C_VEL
LIN {X 0,Y 347.337,Z 606.334,A -85,B 0,C 180,E1 -13758.917,E2 -13758.917} C_VEL
LIN {X 0,Y 346.789,Z 611.796,A -85,B 0,C 180,E1 -13760.67,E2 -13760.67} C_VEL
LIN {X 0,Y 346.461,Z 616.11,A -85,B 0,C 180,E1 -13762.423,E2 -13762.423} C_VEL
LIN {X 0,Y 346.337,Z 619.358,A -85,B 0,C 180,E1 -13764.177,E2 -13764.177} C_VEL
LIN {X 0,Y 346.297,Z 620.949,A -85,B 0,C 180,E1 -13765.344,E2 -13765.344} C_VEL
LIN {X 0,Y 346.397,Z 623.234,A -85,B 0,C 180,E1 -13767.674,E2 -13767.674} C_VEL
LIN {X 0,Y 346.414,Z 624.197,A -85,B 0,C 180,E1 -13768.838,E2 -13768.838} C_VEL
LIN {X 0,Y 346.399,Z 624.74,A -85,B 0,C 180,E1 -13770,E2 -13770} C_VEL
LIN {X 0,Y 346.4,Z 624.872,A -85,B 0,C 180,E1 -13771.163,E2 -13771.163} C_VEL
LIN {X 0,Y 346.272,Z 624.543,A -85,B 0,C 180,E1 -13772.326,E2 -13772.326} C_VEL
LIN {X 0,Y 346.215,Z 623.786,A -85,B 0,C 180,E1 -13773.491,E2 -13773.491} C_VEL
LIN {X 0,Y 346.233,Z 622.625,A -85,B 0,C 180,E1 -13774.657,E2 -13774.657} C_VEL
LIN {X 0,Y 346.242,Z 620.845,A -85,B 0,C 180,E1 -13775.956,E2 -13775.956} C_VEL
LIN {X 0,Y 346.543,Z 616.519,A -85,B 0,C 180,E1 -13778.161,E2 -13778.161} C_VEL
LIN {X 0,Y 346.965,Z 611.913,A -85,B 0,C 180,E1 -13779.914,E2 -13779.914} C_VEL
LIN {X 0,Y 347.817,Z 605.088,A -85,B 0,C 180,E1 -13781.953,E2 -13781.953} C_VEL
LIN {X 0,Y 348.887,Z 597.775,A -85,B 0,C 180,E1 -13783.691,E2 -13783.691} C_VEL
LIN {X 0,Y 350.175,Z 588.757,A -85,B 0,C 180,E1 -13785.451,E2 -13785.451} C_VEL
LIN {X 0,Y 351.978,Z 578.119,A -85,B 0,C 180,E1 -13787.129,E2 -13787.129} C_VEL
LIN {X 0,Y 353.975,Z 565.864,A -85,B 0,C 180,E1 -13788.672,E2 -13788.672} C_VEL
LIN {X 0,Y 354.681,Z 559.374,A -85,B 0,C 180,E1 -13789.384,E2 -13789.384} C_VEL
LIN {X 0,Y 354.763,Z 547.803,A -85,B 0,C 180,E1 -13790.583,E2 -13790.583} C_VEL
LIN {X 0,Y 353.471,Z 536.234,A -85,B 0,C 180,E1 -13791.711,E2 -13791.711} C_VEL
LIN {X 0,Y 350.89,Z 524.205,A -85,B 0,C 180,E1 -13792.877,E2 -13792.877} C_VEL
LIN {X 0,Y 348.409,Z 516.18,A -85,B 0,C 180,E1 -13793.663,E2 -13793.663} C_VEL
LIN {X 0,Y 347.741,Z 513.188,A -85,B 0,C 180,E1 -13793.94,E2 -13793.94} C_VEL
LIN {X 0,Y 348.508,Z 506.681,A -85,B 0,C 180,E1 -13797.634,E2 -13797.634} C_VEL
LIN {X 0,Y 349.533,Z 500.483,A -85,B 0,C 180,E1 -13801.519,E2 -13801.519} C_VEL
LIN {X 0,Y 350.445,Z 496.008,A -85,B 0,C 180,E1 -13804.691,E2 -13804.691} C_VEL
LIN {X 0,Y 350.869,Z 493.249,A -85,B 0,C 180,E1 -13806.935,E2 -13806.935} C_VEL
LIN {X 0,Y 350.879,Z 491.449,A -85,B 0,C 180,E1 -13808.633,E2 -13808.633} C_VEL
LIN {X 0,Y 350.473,Z 488.488,A -85,B 0,C 180,E1 -13812.102,E2 -13812.102} C_VEL
LIN {X 0,Y 350.141,Z 486.452,A -85,B 0,C 180,E1 -13815.371,E2 -13815.371} C_VEL
LIN {X 0,Y 349.863,Z 485.182,A -85,B 0,C 180,E1 -13818.479,E2 -13818.479} C_VEL
LIN {X 0,Y 349.634,Z 484.513,A -85,B 0,C 180,E1 -13821.623,E2 -13821.623} C_VEL
LIN {X 0,Y 349.397,Z 484.393,A -85,B 0,C 180,E1 -13824.315,E2 -13824.315} C_VEL
LIN {X 0,Y 349.005,Z 484.796,A -85,B 0,C 180,E1 -13827.754,E2 -13827.754} C_VEL
LIN {X 0,Y 348.522,Z 485.683,A -85,B 0,C 180,E1 -13831.056,E2 -13831.056} C_VEL
LIN {X 0,Y 348.057,Z 487.19,A -85,B 0,C 180,E1 -13834.911,E2 -13834.911} C_VEL
LIN {X 0,Y 347.955,Z 487.975,A -85,B 0,C 180,E1 -13836.278,E2 -13836.278} C_VEL
LIN {X 0,Y 349.082,Z 490.882,A -85,B 0,C 180,E1 -13836.62,E2 -13836.62} C_VEL
LIN {X 0,Y 350.065,Z 492.672,A -85,B 0,C 180,E1 -13836.876,E2 -13836.876} C_VEL
LIN {X 0,Y 354.719,Z 503.244,A -85,B 0,C 180,E1 -13838.251,E2 -13838.251} C_VEL
LIN {X 0,Y 357.708,Z 513.477,A -85,B 0,C 180,E1 -13839.506,E2 -13839.506} C_VEL
LIN {X 0,Y 358.384,Z 516.831,A -85,B 0,C 180,E1 -13839.915,E2 -13839.915} C_VEL
LIN {X 0,Y 356.847,Z 527.642,A -85,B 0,C 180,E1 -13840.97,E2 -13840.97} C_VEL
LIN {X 0,Y 355.143,Z 538.647,A -85,B 0,C 180,E1 -13842.317,E2 -13842.317} C_VEL
LIN {X 0,Y 353.376,Z 548.883,A -85,B 0,C 180,E1 -13843.833,E2 -13843.833} C_VEL
LIN {X 0,Y 351.89,Z 556.682,A -85,B 0,C 180,E1 -13845.248,E2 -13845.248} C_VEL
LIN {X 0,Y 350.485,Z 564.358,A -85,B 0,C 180,E1 -13846.963,E2 -13846.963} C_VEL
LIN {X 0,Y 349.262,Z 571.565,A -85,B 0,C 180,E1 -13848.98,E2 -13848.98} C_VEL
LIN {X 0,Y 348.332,Z 576.413,A -85,B 0,C 180,E1 -13850.712,E2 -13850.712} C_VEL
LIN {X 0,Y 347.78,Z 579.211,A -85,B 0,C 180,E1 -13851.974,E2 -13851.974} C_VEL
LIN {X 0,Y 347.326,Z 581.16,A -85,B 0,C 180,E1 -13853.027,E2 -13853.027} C_VEL
LIN {X 0,Y 347.064,Z 582.881,A -85,B 0,C 180,E1 -13854.189,E2 -13854.189} C_VEL
LIN {X 0,Y 347,Z 584.138,A -85,B 0,C 180,E1 -13855.353,E2 -13855.353} C_VEL
LIN {X 0,Y 346.778,Z 585.014,A -85,B 0,C 180,E1 -13856.515,E2 -13856.515} C_VEL
LIN {X 0,Y 346.595,Z 585.498,A -85,B 0,C 180,E1 -13857.676,E2 -13857.676} C_VEL
LIN {X 0,Y 346.464,Z 585.579,A -85,B 0,C 180,E1 -13858.838,E2 -13858.838} C_VEL
LIN {X 0,Y 346.402,Z 585.211,A -85,B 0,C 180,E1 -13860,E2 -13860} C_VEL
LIN {X 0,Y 346.406,Z 584.444,A -85,B 0,C 180,E1 -13861.163,E2 -13861.163} C_VEL
LIN {X 0,Y 346.425,Z 583.279,A -85,B 0,C 180,E1 -13862.326,E2 -13862.326} C_VEL
LIN {X 0,Y 346.465,Z 580.708,A -85,B 0,C 180,E1 -13864.072,E2 -13864.072} C_VEL
LIN {X 0,Y 346.691,Z 577.123,A -85,B 0,C 180,E1 -13865.818,E2 -13865.818} C_VEL
LIN {X 0,Y 346.981,Z 572.433,A -85,B 0,C 180,E1 -13867.566,E2 -13867.566} C_VEL
LIN {X 0,Y 347.477,Z 565.339,A -85,B 0,C 180,E1 -13869.606,E2 -13869.606} C_VEL
LIN {X 0,Y 348.116,Z 557.685,A -85,B 0,C 180,E1 -13871.353,E2 -13871.353} C_VEL
LIN {X 0,Y 348.77,Z 549.935,A -85,B 0,C 180,E1 -13872.807,E2 -13872.807} C_VEL
LIN {X 0,Y 349.681,Z 539.547,A -85,B 0,C 180,E1 -13874.402,E2 -13874.402} C_VEL
LIN {X 0,Y 350.545,Z 529.041,A -85,B 0,C 180,E1 -13875.714,E2 -13875.714} C_VEL
LIN {X 0,Y 351.362,Z 517.771,A -85,B 0,C 180,E1 -13876.86,E2 -13876.86} C_VEL
LIN {X 0,Y 352.075,Z 508.197,A -85,B 0,C 180,E1 -13877.648,E2 -13877.648} C_VEL
LIN {X 0,Y 349.528,Z 495.097,A -85,B 0,C 180,E1 -13878.614,E2 -13878.614} C_VEL
LIN {X 0,Y 346.685,Z 481.525,A -85,B 0,C 180,E1 -13879.388,E2 -13879.388} C_VEL
LIN {X 0,Y 346.572,Z 480.711,A -85,B 0,C 180,E1 -13879.472,E2 -13879.472} C_VEL
LIN {X 0,Y 346.603,Z 477.601,A -85,B 0,C 180,E1 -13882.66,E2 -13882.66} C_VEL
LIN {X 0,Y 346.776,Z 473.975,A -85,B 0,C 180,E1 -13886.479,E2 -13886.479} C_VEL
LIN {X 0,Y 346.823,Z 473.289,A -85,B 0,C 180,E1 -13887.78,E2 -13887.78} C_VEL
LIN {X 0,Y 347.128,Z 473.249,A -85,B 0,C 180,E1 -13890.408,E2 -13890.408} C_VEL
LIN {X 0,Y 347.555,Z 473.194,A -85,B 0,C 180,E1 -13894.486,E2 -13894.486} C_VEL
LIN {X 0,Y 347.766,Z 473.166,A -85,B 0,C 180,E1 -13897.987,E2 -13897.987} C_VEL
LIN {X 0,Y 347.754,Z 473.166,A -85,B 0,C 180,E1 -13901.83,E2 -13901.83} C_VEL
LIN {X 0,Y 347.711,Z 473.17,A -85,B 0,C 180,E1 -13905.027,E2 -13905.027} C_VEL
LIN {X 0,Y 347.754,Z 473.169,A -85,B 0,C 180,E1 -13908.397,E2 -13908.397} C_VEL
LIN {X 0,Y 347.781,Z 473.165,A -85,B 0,C 180,E1 -13912.011,E2 -13912.011} C_VEL
LIN {X 0,Y 347.748,Z 473.166,A -85,B 0,C 180,E1 -13915.536,E2 -13915.536} C_VEL
LIN {X 0,Y 347.768,Z 473.164,A -85,B 0,C 180,E1 -13919.654,E2 -13919.654} C_VEL
LIN {X 0,Y 347.856,Z 473.153,A -85,B 0,C 180,E1 -13922.745,E2 -13922.745} C_VEL
LIN {X 0,Y 347.793,Z 473.165,A -85,B 0,C 180,E1 -13926.162,E2 -13926.162} C_VEL
LIN {X 0,Y 347.822,Z 473.16,A -85,B 0,C 180,E1 -13929.91,E2 -13929.91} C_VEL
LIN {X 0,Y 347.871,Z 473.154,A -85,B 0,C 180,E1 -13932.359,E2 -13932.359} C_VEL
LIN {X 0,Y 347.902,Z 473.151,A -85,B 0,C 180,E1 -13935.971,E2 -13935.971} C_VEL
LIN {X 0,Y 347.933,Z 473.143,A -85,B 0,C 180,E1 -13939.526,E2 -13939.526} C_VEL
LIN {X 0,Y 348.08,Z 473.128,A -85,B 0,C 180,E1 -13941.875,E2 -13941.875} C_VEL
LIN {X 0,Y 348.073,Z 473.129,A -85,B 0,C 180,E1 -13944.206,E2 -13944.206} C_VEL
LIN {X 0,Y 348.211,Z 473.111,A -85,B 0,C 180,E1 -13947.687,E2 -13947.687} C_VEL
LIN {X 0,Y 348.35,Z 473.096,A -85,B 0,C 180,E1 -13950,E2 -13950} C_VEL
LIN {X 0,Y 348.211,Z 473.11,A -85,B 0,C 180,E1 -13952.313,E2 -13952.313} C_VEL
LIN {X 0,Y 348.073,Z 473.125,A -85,B 0,C 180,E1 -13956.958,E2 -13956.958} C_VEL
LIN {X 0,Y 347.932,Z 473.144,A -85,B 0,C 180,E1 -13960.474,E2 -13960.474} C_VEL
LIN {X 0,Y 347.903,Z 473.149,A -85,B 0,C 180,E1 -13964.15,E2 -13964.15} C_VEL
LIN {X 0,Y 347.896,Z 473.149,A -85,B 0,C 180,E1 -13968.29,E2 -13968.29} C_VEL
LIN {X 0,Y 347.78,Z 473.165,A -85,B 0,C 180,E1 -13971.63,E2 -13971.63} C_VEL
LIN {X 0,Y 347.815,Z 473.157,A -85,B 0,C 180,E1 -13975.108,E2 -13975.108} C_VEL
LIN {X 0,Y 347.812,Z 473.161,A -85,B 0,C 180,E1 -13977.694,E2 -13977.694} C_VEL
LIN {X 0,Y 347.753,Z 473.166,A -85,B 0,C 180,E1 -13980.348,E2 -13980.348} C_VEL
LIN {X 0,Y 347.752,Z 473.169,A -85,B 0,C 180,E1 -13984.044,E2 -13984.044} C_VEL
LIN {X 0,Y 347.77,Z 473.164,A -85,B 0,C 180,E1 -13987.32,E2 -13987.32} C_VEL
LIN {X 0,Y 347.737,Z 473.168,A -85,B 0,C 180,E1 -13990.297,E2 -13990.297} C_VEL
LIN {X 0,Y 347.727,Z 473.171,A -85,B 0,C 180,E1 -13993.408,E2 -13993.408} C_VEL
LIN {X 0,Y 347.729,Z 473.168,A -85,B 0,C 180,E1 -13996.686,E2 -13996.686} C_VEL
LIN {X 0,Y 347.751,Z 473.166,A -85,B 0,C 180,E1 -14000.173,E2 -14000.173} C_VEL
LIN {X 0,Y 347.753,Z 473.164,A -85,B 0,C 180,E1 -14002.677,E2 -14002.677} C_VEL
LIN {X 0,Y 347.617,Z 473.186,A -85,B 0,C 180,E1 -14005.559,E2 -14005.559} C_VEL
LIN {X 0,Y 346.881,Z 473.275,A -85,B 0,C 180,E1 -14006.525,E2 -14006.525} C_VEL
LIN {X 0,Y 343.871,Z 473.651,A -85,B 0,C 180,E1 -14008.091,E2 -14008.091} C_VEL
LIN {X 0,Y 341.296,Z 473.972,A -85,B 0,C 180,E1 -14009.359,E2 -14009.359} C_VEL
LIN {X 0,Y 340.127,Z 474.116,A -85,B 0,C 180,E1 -14010.343,E2 -14010.343} C_VEL
LIN {X 0,Y 339.997,Z 474.131,A -85,B 0,C 180,E1 -14010.677,E2 -14010.677} C_VEL
LIN {X 0,Y 339.753,Z 474.163,A -85,B 0,C 180,E1 -14012.929,E2 -14012.929} C_VEL
LIN {X 0,Y 339.487,Z 474.33,A -85,B 0,C 180,E1 -14014.724,E2 -14014.724} C_VEL
LIN {X 0,Y 339.477,Z 478.582,A -85,B 0,C 180,E1 -14018.688,E2 -14018.688} C_VEL
LIN {X 0,Y 339.447,Z 480.504,A -85,B 0,C 180,E1 -14020.457,E2 -14020.457} C_VEL
LIN {X 0,Y 342.314,Z 494.814,A -85,B 0,C 180,E1 -14021.261,E2 -14021.261} C_VEL
LIN {X 0,Y 344.945,Z 508.302,A -85,B 0,C 180,E1 -14022.281,E2 -14022.281} C_VEL
LIN {X 0,Y 344.15,Z 521.018,A -85,B 0,C 180,E1 -14023.387,E2 -14023.387} C_VEL
LIN {X 0,Y 343.248,Z 533.021,A -85,B 0,C 180,E1 -14024.715,E2 -14024.715} C_VEL
LIN {X 0,Y 342.372,Z 542.76,A -85,B 0,C 180,E1 -14026.042,E2 -14026.042} C_VEL
LIN {X 0,Y 341.365,Z 553.316,A -85,B 0,C 180,E1 -14027.817,E2 -14027.817} C_VEL
LIN {X 0,Y 340.656,Z 561.833,A -85,B 0,C 180,E1 -14029.6,E2 -14029.6} C_VEL
LIN {X 0,Y 339.993,Z 569.736,A -85,B 0,C 180,E1 -14031.68,E2 -14031.68} C_VEL
LIN {X 0,Y 339.609,Z 575.702,A -85,B 0,C 180,E1 -14033.727,E2 -14033.727} C_VEL
LIN {X 0,Y 339.39,Z 580.31,A -85,B 0,C 180,E1 -14035.843,E2 -14035.843} C_VEL
LIN {X 0,Y 339.321,Z 583.044,A -85,B 0,C 180,E1 -14037.626,E2 -14037.626} C_VEL
LIN {X 0,Y 339.29,Z 584.333,A -85,B 0,C 180,E1 -14038.813,E2 -14038.813} C_VEL
LIN {X 0,Y 339.313,Z 585.172,A -85,B 0,C 180,E1 -14040,E2 -14040} C_VEL
LIN {X 0,Y 339.387,Z 585.618,A -85,B 0,C 180,E1 -14041.186,E2 -14041.186} C_VEL
LIN {X 0,Y 339.531,Z 585.664,A -85,B 0,C 180,E1 -14042.372,E2 -14042.372} C_VEL
LIN {X 0,Y 339.731,Z 585.262,A -85,B 0,C 180,E1 -14043.558,E2 -14043.558} C_VEL
LIN {X 0,Y 339.891,Z 584.47,A -85,B 0,C 180,E1 -14044.744,E2 -14044.744} C_VEL
LIN {X 0,Y 339.945,Z 583.305,A -85,B 0,C 180,E1 -14045.933,E2 -14045.933} C_VEL
LIN {X 0,Y 340.719,Z 580.046,A -85,B 0,C 180,E1 -14048.069,E2 -14048.069} C_VEL
LIN {X 0,Y 341.579,Z 575.646,A -85,B 0,C 180,E1 -14050.072,E2 -14050.072} C_VEL
LIN {X 0,Y 342.631,Z 570.599,A -85,B 0,C 180,E1 -14051.836,E2 -14051.836} C_VEL
LIN {X 0,Y 343.814,Z 564.321,A -85,B 0,C 180,E1 -14053.596,E2 -14053.596} C_VEL
LIN {X 0,Y 345.282,Z 556.542,A -85,B 0,C 180,E1 -14055.343,E2 -14055.343} C_VEL
LIN {X 0,Y 347.212,Z 546.989,A -85,B 0,C 180,E1 -14057.067,E2 -14057.067} C_VEL
LIN {X 0,Y 349.05,Z 536.631,A -85,B 0,C 180,E1 -14058.582,E2 -14058.582} C_VEL
LIN {X 0,Y 350.877,Z 525.372,A -85,B 0,C 180,E1 -14059.908,E2 -14059.908} C_VEL
LIN {X 0,Y 351.918,Z 518.47,A -85,B 0,C 180,E1 -14060.583,E2 -14060.583} C_VEL
LIN {X 0,Y 351.36,Z 514.203,A -85,B 0,C 180,E1 -14061.103,E2 -14061.103} C_VEL
LIN {X 0,Y 349.109,Z 505.838,A -85,B 0,C 180,E1 -14062.174,E2 -14062.174} C_VEL
LIN {X 0,Y 345.029,Z 495.485,A -85,B 0,C 180,E1 -14063.563,E2 -14063.563} C_VEL
LIN {X 0,Y 342.328,Z 489.886,A -85,B 0,C 180,E1 -14064.343,E2 -14064.343} C_VEL
LIN {X 0,Y 341.069,Z 486.99,A -85,B 0,C 180,E1 -14064.736,E2 -14064.736} C_VEL
LIN {X 0,Y 340.999,Z 486.599,A -85,B 0,C 180,E1 -14064.804,E2 -14064.804} C_VEL
LIN {X 0,Y 341.176,Z 483.664,A -85,B 0,C 180,E1 -14068.28,E2 -14068.28} C_VEL
LIN {X 0,Y 341.393,Z 481.484,A -85,B 0,C 180,E1 -14070.974,E2 -14070.974} C_VEL
LIN {X 0,Y 341.523,Z 479.429,A -85,B 0,C 180,E1 -14073.753,E2 -14073.753} C_VEL
LIN {X 0,Y 341.428,Z 477.562,A -85,B 0,C 180,E1 -14076.651,E2 -14076.651} C_VEL
LIN {X 0,Y 341.173,Z 476.068,A -85,B 0,C 180,E1 -14079.686,E2 -14079.686} C_VEL
LIN {X 0,Y 340.848,Z 474.95,A -85,B 0,C 180,E1 -14082.877,E2 -14082.877} C_VEL
LIN {X 0,Y 340.854,Z 474.555,A -85,B 0,C 180,E1 -14085.286,E2 -14085.286} C_VEL
LIN {X 0,Y 341.848,Z 480.172,A -85,B 0,C 180,E1 -14088.861,E2 -14088.861} C_VEL
LIN {X 0,Y 342.739,Z 485.397,A -85,B 0,C 180,E1 -14092.036,E2 -14092.036} C_VEL
LIN {X 0,Y 342.977,Z 487.972,A -85,B 0,C 180,E1 -14093.541,E2 -14093.541} C_VEL
LIN {X 0,Y 342.495,Z 493.012,A -85,B 0,C 180,E1 -14096.355,E2 -14096.355} C_VEL
LIN {X 0,Y 341.579,Z 500.483,A -85,B 0,C 180,E1 -14100.409,E2 -14100.409} C_VEL
LIN {X 0,Y 340.87,Z 506.649,A -85,B 0,C 180,E1 -14103.686,E2 -14103.686} C_VEL
LIN {X 0,Y 340.6,Z 509.781,A -85,B 0,C 180,E1 -14105.332,E2 -14105.332} C_VEL
LIN {X 0,Y 341.339,Z 513.646,A -85,B 0,C 180,E1 -14105.683,E2 -14105.683} C_VEL
LIN {X 0,Y 342.104,Z 515.922,A -85,B 0,C 180,E1 -14105.923,E2 -14105.923} C_VEL
LIN {X 0,Y 345.142,Z 528.422,A -85,B 0,C 180,E1 -14107.152,E2 -14107.152} C_VEL
LIN {X 0,Y 347.009,Z 539.867,A -85,B 0,C 180,E1 -14108.297,E2 -14108.297} C_VEL
LIN {X 0,Y 347.674,Z 549.622,A -85,B 0,C 180,E1 -14109.308,E2 -14109.308} C_VEL
LIN {X 0,Y 347.447,Z 562.983,A -85,B 0,C 180,E1 -14110.81,E2 -14110.81} C_VEL
LIN {X 0,Y 345.674,Z 573.372,A -85,B 0,C 180,E1 -14112.091,E2 -14112.091} C_VEL
LIN {X 0,Y 343.939,Z 583.938,A -85,B 0,C 180,E1 -14113.693,E2 -14113.693} C_VEL
LIN {X 0,Y 342.605,Z 591.869,A -85,B 0,C 180,E1 -14115.142,E2 -14115.142} C_VEL
LIN {X 0,Y 341.385,Z 599.877,A -85,B 0,C 180,E1 -14116.912,E2 -14116.912} C_VEL
LIN {X 0,Y 340.353,Z 606.47,A -85,B 0,C 180,E1 -14118.687,E2 -14118.687} C_VEL
LIN {X 0,Y 339.744,Z 611.785,A -85,B 0,C 180,E1 -14120.474,E2 -14120.474} C_VEL
LIN {X 0,Y 339.39,Z 615.969,A -85,B 0,C 180,E1 -14122.264,E2 -14122.264} C_VEL
LIN {X 0,Y 339.258,Z 619.129,A -85,B 0,C 180,E1 -14124.055,E2 -14124.055} C_VEL
LIN {X 0,Y 339.213,Z 620.665,A -85,B 0,C 180,E1 -14125.246,E2 -14125.246} C_VEL
LIN {X 0,Y 339.353,Z 623.645,A -85,B 0,C 180,E1 -14128.813,E2 -14128.813} C_VEL
LIN {X 0,Y 339.338,Z 624.231,A -85,B 0,C 180,E1 -14130,E2 -14130} C_VEL
LIN {X 0,Y 339.335,Z 624.403,A -85,B 0,C 180,E1 -14131.187,E2 -14131.187} C_VEL
LIN {X 0,Y 339.175,Z 624.149,A -85,B 0,C 180,E1 -14132.375,E2 -14132.375} C_VEL
LIN {X 0,Y 339.136,Z 623.445,A -85,B 0,C 180,E1 -14133.564,E2 -14133.564} C_VEL
LIN {X 0,Y 339.129,Z 622.326,A -85,B 0,C 180,E1 -14134.755,E2 -14134.755} C_VEL
LIN {X 0,Y 339.141,Z 620.8,A -85,B 0,C 180,E1 -14135.947,E2 -14135.947} C_VEL
LIN {X 0,Y 339.38,Z 617.682,A -85,B 0,C 180,E1 -14137.736,E2 -14137.736} C_VEL
LIN {X 0,Y 339.772,Z 613.539,A -85,B 0,C 180,E1 -14139.525,E2 -14139.525} C_VEL
